C01811=1033.680,159.526,-103.122,169.533,42.942,158.097
C01812=1033.686,159.775,-103.145,169.536,42.941,158.097
C01813=1033.692,160.024,-103.167,169.539,42.940,158.097
C01814=1033.698,160.273,-103.190,169.542,42.939,158.097
C01815=1033.703,160.521,-103.212,169.544,42.939,158.097
C01816=1033.709,160.770,-103.235,169.547,42.938,158.097
C01817=1033.715,161.019,-103.257,169.550,42.937,158.097
C01818=1033.721,161.268,-103.280,169.553,42.936,158.097
C01819=1033.727,161.517,-103.303,169.556,42.935,158.097
C01820=1033.732,161.766,-103.326,169.559,42.934,158.097
C01821=1033.739,162.014,-103.348,169.561,42.933,158.097
C01822=1033.744,162.264,-103.370,169.564,42.933,158.097
C01823=1033.750,162.513,-103.393,169.566,42.932,158.097
C01824=1033.756,162.762,-103.416,169.569,42.931,158.097
C01825=1033.762,163.010,-103.438,169.572,42.930,158.097
C01826=1033.768,163.259,-103.461,169.575,42.930,158.097
C01827=1033.774,163.508,-103.484,169.577,42.929,158.097
C01828=1033.779,163.757,-103.507,169.580,42.928,158.098
C01829=1033.786,164.006,-103.530,169.583,42.927,158.098
C01830=1033.791,164.254,-103.552,169.586,42.926,158.098
C01831=1033.797,164.504,-103.575,169.589,42.925,158.098
C01832=1033.803,164.753,-103.598,169.592,42.924,158.098
C01833=1033.809,165.001,-103.620,169.595,42.924,158.098
C01834=1033.815,165.250,-103.643,169.598,42.922,158.098
C01835=1033.821,165.499,-103.666,169.600,42.922,158.098
C01836=1033.826,165.748,-103.689,169.603,42.921,158.098
C01837=1033.833,165.997,-103.711,169.606,42.920,158.098
C01838=1033.839,166.246,-103.735,169.608,42.919,158.098
C01839=1033.845,166.495,-103.757,169.611,42.918,158.098
C01840=1033.851,166.744,-103.780,169.614,42.918,158.098
C01841=1033.856,166.993,-103.803,169.617,42.916,158.098
C01842=1033.863,167.242,-103.826,169.620,42.916,158.098
C01843=1033.868,167.491,-103.849,169.623,42.915,158.098
C01844=1033.874,167.739,-103.872,169.626,42.914,158.098
C01845=1033.880,167.988,-103.895,169.628,42.913,158.098
C01846=1033.886,168.237,-103.917,169.631,42.913,158.098
C01847=1033.892,168.486,-103.940,169.634,42.912,158.098
C01848=1033.898,168.735,-103.963,169.637,42.911,158.098
C01849=1033.905,168.984,-103.987,169.640,42.910,158.098
C01850=1033.910,169.233,-104.010,169.643,42.910,158.098
C01851=1033.917,169.481,-104.032,169.645,42.908,158.098
C01852=1033.922,169.730,-104.055,169.649,42.908,158.099
C01853=1033.928,169.979,-104.078,169.651,42.907,158.099
C01854=1033.934,170.228,-104.101,169.654,42.906,158.099
C01855=1033.940,170.477,-104.124,169.657,42.905,158.099
C01856=1033.947,170.726,-104.147,169.660,42.904,158.099
C01857=1033.953,170.974,-104.170,169.663,42.903,158.099
C01858=1033.958,171.223,-104.193,169.666,42.902,158.099
C01859=1033.964,171.472,-104.216,169.669,42.902,158.099
C01860=1033.970,171.721,-104.239,169.672,42.901,158.099
C01861=1033.976,171.971,-104.262,169.675,42.900,158.099
C01862=1033.983,172.219,-104.285,169.678,42.899,158.099
C01863=1033.989,172.503,-104.312,169.681,42.898,158.099
C01864=1033.996,172.787,-104.338,169.684,42.897,158.099
C01865=1034.004,173.072,-104.364,169.688,42.897,158.099
C01866=1034.010,173.356,-104.391,169.690,42.896,158.099
C01867=1034.016,173.605,-104.414,169.693,42.894,158.099
C01868=1034.023,173.854,-104.436,169.696,42.894,158.099
C01869=1034.029,174.103,-104.461,169.699,42.893,158.099
C01870=1034.035,174.352,-104.483,169.702,42.892,158.099
C01871=1034.041,174.601,-104.506,169.705,42.891,158.099
C01872=1034.046,174.850,-104.529,169.708,42.891,158.100
C01873=1034.054,175.098,-104.553,169.711,42.889,158.100
C01874=1034.059,175.347,-104.576,169.714,42.889,158.100
C01875=1034.065,175.596,-104.599,169.717,42.888,158.100
C01876=1034.072,175.845,-104.623,169.720,42.887,158.100
C01877=1034.078,176.094,-104.646,169.723,42.886,158.100
C01878=1034.083,176.343,-104.669,169.726,42.886,158.100
C01879=1034.090,176.591,-104.692,169.729,42.884,158.100
C01880=1034.096,176.840,-104.715,169.732,42.884,158.100
C01881=1034.102,177.089,-104.739,169.735,42.883,158.100
C01882=1034.108,177.338,-104.762,169.738,42.882,158.100
C01883=1034.114,177.587,-104.785,169.741,42.882,158.100
C01884=1034.121,177.835,-104.809,169.744,42.881,158.100
C01885=1034.126,178.084,-104.831,169.747,42.880,158.100
C01886=1034.134,178.333,-104.855,169.750,42.879,158.100
C01887=1034.139,178.582,-104.878,169.753,42.878,158.100
C01888=1034.146,178.832,-104.901,169.756,42.877,158.100
C01889=1034.152,179.080,-104.925,169.759,42.877,158.101
C01890=1034.157,179.329,-104.948,169.762,42.876,158.101
C01891=1034.164,179.578,-104.972,169.765,42.875,158.101
C01892=1034.171,179.826,-104.994,169.768,42.874,158.101
C01893=1034.177,180.075,-105.018,169.771,42.873,158.101
C01894=1034.183,180.324,-105.041,169.774,42.872,158.101
C01895=1034.189,180.572,-105.065,169.777,42.872,158.101
C01896=1034.195,180.822,-105.088,169.780,42.871,158.101
C01897=1034.201,181.070,-105.112,169.783,42.870,158.101
C01898=1034.208,181.320,-105.135,169.787,42.869,158.101
C01899=1034.214,181.568,-105.159,169.790,42.868,158.101
C01900=1034.221,181.817,-105.182,169.793,42.868,158.101
C01901=1034.227,182.066,-105.205,169.795,42.867,158.101
C01902=1034.233,182.314,-105.229,169.798,42.866,158.101
C01903=1034.239,182.564,-105.252,169.801,42.865,158.101
C01904=1034.245,182.812,-105.276,169.804,42.865,158.101
C01905=1034.252,183.061,-105.300,169.807,42.864,158.102
C01906=1034.258,183.310,-105.323,169.810,42.863,158.101
C01907=1034.264,183.559,-105.347,169.813,42.862,158.102
C01908=1034.270,183.807,-105.371,169.817,42.862,158.102
C01909=1034.276,184.056,-105.395,169.820,42.861,158.102
C01910=1034.281,184.305,-105.419,169.823,42.861,158.102
C01911=1034.287,184.554,-105.442,169.826,42.860,158.102
C01912=1034.293,184.803,-105.467,169.829,42.859,158.102
C01913=1034.299,185.051,-105.491,169.832,42.859,158.102
C01914=1034.305,185.300,-105.514,169.835,42.858,158.102
C01915=1034.311,185.549,-105.539,169.838,42.858,158.102
C01916=1034.317,185.797,-105.562,169.841,42.857,158.103
C01917=1034.323,186.046,-105.587,169.844,42.857,158.103
C01918=1034.329,186.295,-105.611,169.848,42.856,158.103
C01919=1034.335,186.544,-105.635,169.851,42.856,158.103
C01920=1034.341,186.792,-105.659,169.854,42.855,158.103
C01921=1034.346,187.041,-105.683,169.857,42.855,158.103
C01922=1034.353,187.290,-105.707,169.859,42.853,158.103
C01923=1034.358,187.539,-105.731,169.863,42.853,158.103
C01924=1034.365,187.788,-105.755,169.867,42.852,158.103
C01925=1034.371,188.036,-105.779,169.870,42.852,158.104
C01926=1034.376,188.286,-105.803,169.873,42.851,158.104
C01927=1034.383,188.569,-105.831,169.876,42.851,158.104
C01928=1034.390,188.853,-105.859,169.880,42.850,158.104
C01929=1034.397,189.137,-105.886,169.883,42.850,158.104
C01930=1034.404,189.421,-105.914,169.887,42.849,158.104
C01931=1034.410,189.670,-105.938,169.890,42.848,158.104
C01932=1034.416,189.919,-105.962,169.893,42.848,158.105
C01933=1034.422,190.168,-105.986,169.896,42.847,158.105
C01934=1034.428,190.416,-106.010,169.899,42.846,158.105
C01935=1034.434,190.665,-106.034,169.903,42.846,158.105
C01936=1034.440,190.914,-106.059,169.906,42.845,158.105
C01937=1034.447,191.162,-106.083,169.909,42.845,158.105
C01938=1034.452,191.411,-106.108,169.912,42.844,158.105
C01939=1034.459,191.660,-106.132,169.915,42.844,158.105
C01940=1034.464,191.909,-106.156,169.918,42.843,158.105
C01941=1034.470,192.157,-106.180,169.921,42.843,158.106
C01942=1034.476,192.406,-106.204,169.925,42.842,158.106
C01943=1034.483,192.654,-106.229,169.928,42.841,158.106
C01944=1034.489,192.903,-106.253,169.931,42.841,158.106
C01945=1034.495,193.152,-106.277,169.934,42.840,158.106
C01946=1034.501,193.401,-106.302,169.937,42.840,158.106
C01947=1034.507,193.650,-106.326,169.940,42.839,158.106
C01948=1034.513,193.899,-106.351,169.944,42.839,158.106
C01949=1034.519,194.147,-106.375,169.947,42.838,158.107
C01950=1034.525,194.396,-106.399,169.950,42.838,158.107
C01951=1034.532,194.645,-106.423,169.954,42.837,158.107
C01952=1034.538,194.893,-106.448,169.957,42.837,158.107
C01953=1034.544,195.142,-106.472,169.961,42.836,158.107
C01954=1034.550,195.391,-106.497,169.964,42.836,158.107
C01955=1034.556,195.639,-106.521,169.967,42.835,158.107
C01956=1034.562,195.888,-106.546,169.970,42.835,158.107
C01957=1034.569,196.137,-106.570,169.973,42.834,158.108
C01958=1034.575,196.385,-106.595,169.977,42.833,158.108
C01959=1034.581,196.634,-106.619,169.980,42.833,158.108
C01960=1034.587,196.884,-106.644,169.983,42.832,158.108
C01961=1034.593,197.131,-106.668,169.986,42.832,158.108
C01962=1034.599,197.381,-106.693,169.990,42.831,158.108
C01963=1034.606,197.630,-106.717,169.993,42.831,158.108
C01964=1034.612,197.878,-106.742,169.996,42.830,158.109
C01965=1034.618,198.126,-106.766,169.999,42.830,158.109
C01966=1034.624,198.375,-106.791,170.003,42.829,158.109
C01967=1034.630,198.624,-106.816,170.006,42.829,158.109
C01968=1034.637,198.873,-106.840,170.009,42.828,158.109
C01969=1034.643,199.122,-106.865,170.012,42.828,158.109
C01970=1034.649,199.370,-106.889,170.016,42.827,158.109
C01971=1034.655,199.619,-106.914,170.019,42.826,158.109
C01972=1034.662,199.868,-106.938,170.023,42.827,158.110
C01973=1034.668,200.117,-106.963,170.026,42.826,158.110
C01974=1034.675,200.366,-106.987,170.030,42.825,158.110
C01975=1034.681,200.614,-107.012,170.033,42.825,158.110
C01976=1034.687,200.862,-107.038,170.036,42.824,158.110
C01977=1034.693,201.112,-107.062,170.039,42.824,158.110
C01978=1034.700,201.360,-107.087,170.043,42.824,158.111
C01979=1034.705,201.609,-107.112,170.046,42.823,158.111
C01980=1034.711,201.857,-107.137,170.049,42.823,158.111
C01981=1034.717,202.106,-107.162,170.052,42.822,158.111
C01982=1034.723,202.354,-107.187,170.056,42.822,158.111
C01983=1034.729,202.604,-107.212,170.059,42.822,158.111
C01984=1034.736,202.852,-107.237,170.062,42.821,158.112
C01985=1034.741,203.100,-107.262,170.067,42.821,158.112
C01986=1034.747,203.350,-107.287,170.070,42.821,158.112
C01987=1034.754,203.598,-107.312,170.073,42.820,158.112
C01988=1034.760,203.847,-107.337,170.076,42.820,158.112
C01989=1034.766,204.095,-107.362,170.080,42.820,158.113
C01990=1034.773,204.344,-107.388,170.083,42.819,158.113
C01991=1034.798,205.393,-107.493,170.407,42.924,158.158
C01992=1034.808,205.731,-107.529,170.411,42.924,158.159
C01993=1034.817,206.069,-107.565,170.414,42.925,158.159
C01994=1034.826,206.405,-107.600,170.417,42.925,158.159
C01995=1034.835,206.743,-107.636,170.421,42.925,158.160
C01996=1034.842,206.992,-107.663,170.423,42.926,158.160
C01997=1034.848,207.240,-107.689,170.425,42.927,158.160
C01998=1034.855,207.489,-107.716,170.427,42.927,158.160
C01999=1034.862,207.737,-107.742,170.430,42.927,158.161
C02000=1034.869,207.985,-107.768,170.432,42.928,158.161
C02001=1034.875,208.235,-107.795,170.435,42.928,158.161
C02002=1034.882,208.483,-107.821,170.438,42.929,158.162
C02003=1034.889,208.731,-107.848,170.440,42.929,158.162
C02004=1034.896,208.979,-107.875,170.442,42.929,158.162
C02005=1034.902,209.228,-107.902,170.445,42.930,158.162
C02006=1034.909,209.477,-107.928,170.448,42.930,158.163
C02007=1034.916,209.725,-107.954,170.450,42.931,158.163
C02008=1034.922,209.974,-107.981,170.452,42.931,158.163
C02009=1034.929,210.222,-108.007,170.455,42.932,158.163
C02010=1034.936,210.470,-108.034,170.457,42.932,158.164
C02011=1034.942,210.719,-108.061,170.460,42.932,158.164
C02012=1034.950,210.968,-108.088,170.463,42.933,158.164
C02013=1034.956,211.216,-108.114,170.465,42.933,158.165
C02014=1034.962,211.465,-108.141,170.467,42.934,158.165
C02015=1034.970,211.713,-108.168,170.469,42.934,158.165
C02016=1034.976,211.961,-108.195,170.473,42.935,158.165
C02017=1034.983,212.210,-108.221,170.475,42.935,158.166
C02018=1034.989,212.458,-108.249,170.477,42.935,158.166
C02019=1034.996,212.707,-108.275,170.480,42.936,158.166
C02020=1035.002,212.956,-108.302,170.482,42.936,158.166
C02021=1035.010,213.204,-108.329,170.485,42.937,158.167
C02022=1035.015,213.452,-108.356,170.488,42.938,158.167
C02023=1035.022,213.701,-108.383,170.490,42.938,158.167
C02024=1035.029,213.949,-108.410,170.492,42.938,158.168
C02025=1035.036,214.198,-108.437,170.494,42.939,158.168
C02026=1035.042,214.446,-108.463,170.498,42.939,158.168
C02027=1035.049,214.695,-108.490,170.500,42.939,158.168
C02028=1035.056,214.944,-108.517,170.502,42.940,158.169
C02029=1035.062,215.191,-108.544,170.505,42.941,158.169
C02030=1035.069,215.440,-108.571,170.508,42.941,158.169
C02031=1035.076,215.688,-108.598,170.510,42.942,158.170
C02032=1035.083,215.937,-108.625,170.513,42.942,158.170
C02033=1035.089,216.185,-108.652,170.515,42.942,158.170
C02034=1035.096,216.434,-108.679,170.518,42.943,158.171
C02035=1035.103,216.683,-108.706,170.520,42.943,158.171
C02036=1035.110,216.931,-108.733,170.523,42.944,158.171
C02037=1035.116,217.180,-108.760,170.525,42.944,158.171
C02038=1035.123,217.427,-108.787,170.528,42.945,158.172
C02039=1035.130,217.676,-108.814,170.531,42.945,158.172
C02040=1035.137,217.925,-108.841,170.533,42.945,158.172
C02041=1035.143,218.174,-108.868,170.536,42.946,158.173
C02042=1035.150,218.422,-108.895,170.539,42.946,158.173
C02043=1035.157,218.670,-108.922,170.541,42.947,158.173
C02044=1035.163,218.919,-108.949,170.543,42.947,158.173
C02045=1035.171,219.167,-108.976,170.546,42.948,158.174
C02046=1035.177,219.416,-109.003,170.549,42.948,158.174
C02047=1035.184,219.664,-109.031,170.551,42.949,158.174
C02048=1035.193,220.007,-109.068,170.556,42.949,158.175
C02049=1035.202,220.349,-109.106,170.559,42.950,158.175
C02050=1035.212,220.693,-109.144,170.562,42.951,158.176
C02051=1035.220,221.036,-109.181,170.566,42.952,158.176
C02052=1035.227,221.284,-109.209,170.568,42.952,158.176
C02053=1035.234,221.532,-109.236,170.571,42.952,158.176
C02054=1035.241,221.781,-109.263,170.574,42.953,158.177
C02055=1035.247,222.029,-109.290,170.576,42.953,158.177
C02056=1035.254,222.277,-109.318,170.579,42.954,158.177
C02057=1035.260,222.526,-109.346,170.582,42.954,158.178
C02058=1035.267,222.775,-109.373,170.584,42.955,158.178
C02059=1035.273,223.023,-109.400,170.586,42.955,158.178
C02060=1035.281,223.271,-109.428,170.590,42.956,158.179
C02061=1035.287,223.520,-109.455,170.592,42.956,158.179
C02062=1035.293,223.768,-109.482,170.594,42.957,158.179
C02063=1035.300,224.017,-109.510,170.598,42.957,158.180
C02064=1035.307,224.265,-109.537,170.600,42.958,158.180
C02065=1035.314,224.513,-109.565,170.602,42.959,158.180
C02066=1035.321,224.762,-109.592,170.606,42.959,158.180
C02067=1035.327,225.010,-109.620,170.608,42.959,158.181
C02068=1035.334,225.259,-109.647,170.610,42.960,158.181
C02069=1035.340,225.508,-109.675,170.614,42.960,158.181
C02070=1035.347,225.756,-109.702,170.616,42.961,158.182
C02071=1035.355,226.004,-109.730,170.618,42.961,158.182
C02072=1035.361,226.253,-109.757,170.622,42.962,158.182
C02073=1035.367,226.500,-109.785,170.624,42.962,158.183
C02074=1035.374,226.749,-109.812,170.627,42.962,158.183
C02075=1035.381,226.997,-109.840,170.630,42.963,158.183
C02076=1035.387,227.246,-109.868,170.632,42.964,158.183
C02077=1035.395,227.494,-109.895,170.635,42.964,158.184
C02078=1035.401,227.742,-109.923,170.638,42.965,158.184
C02079=1035.408,227.991,-109.950,170.640,42.966,158.184
C02080=1035.415,228.239,-109.978,170.643,42.966,158.185
C02081=1035.421,228.488,-110.006,170.646,42.967,158.185
C02082=1035.428,228.736,-110.034,170.649,42.967,158.185
C02083=1035.435,228.985,-110.061,170.651,42.968,158.186
C02084=1035.442,229.233,-110.089,170.654,42.968,158.186
C02085=1035.448,229.481,-110.117,170.657,42.969,158.186
C02086=1035.455,229.730,-110.145,170.659,42.969,158.187
C02087=1035.461,229.979,-110.173,170.662,42.970,158.187
C02088=1035.467,230.227,-110.201,170.665,42.970,158.187
C02089=1035.474,230.475,-110.228,170.667,42.971,158.188
C02090=1035.481,230.723,-110.257,170.671,42.972,158.188
C02091=1035.488,230.972,-110.285,170.673,42.972,158.188
C02092=1035.495,231.220,-110.312,170.676,42.973,158.189
C02093=1035.501,231.469,-110.340,170.679,42.973,158.189
C02094=1035.508,231.717,-110.368,170.681,42.974,158.189
C02095=1035.515,231.966,-110.395,170.685,42.974,158.190
C02096=1035.521,232.214,-110.425,170.687,42.975,158.190
C02097=1035.527,232.462,-110.452,170.689,42.976,158.190
C02098=1035.534,232.711,-110.480,170.693,42.976,158.191
C02099=1035.541,232.959,-110.508,170.695,42.977,158.191
C02100=1035.548,233.207,-110.536,170.698,42.977,158.191
C02101=1035.554,233.456,-110.564,170.701,42.978,158.192
C02102=1035.560,233.704,-110.592,170.703,42.979,158.192
C02103=1035.567,233.952,-110.621,170.706,42.979,158.192
C02104=1035.576,234.288,-110.658,170.710,42.980,158.193
C02105=1035.585,234.623,-110.697,170.714,42.981,158.193
C02106=1035.594,234.958,-110.735,170.718,42.981,158.194
C02107=1035.604,235.293,-110.772,170.721,42.982,158.194
C02108=1035.610,235.542,-110.801,170.724,42.983,158.194
C02109=1035.616,235.790,-110.828,170.727,42.983,158.195
C02110=1035.623,236.038,-110.857,170.730,42.984,158.195
C02111=1035.631,236.287,-110.885,170.733,42.984,158.195
C02112=1035.636,236.536,-110.913,170.735,42.985,158.196
C02113=1035.643,236.784,-110.942,170.739,42.986,158.196
C02114=1035.650,237.032,-110.969,170.741,42.986,158.196
C02115=1035.657,237.280,-110.998,170.744,42.987,158.197
C02116=1035.663,237.529,-111.026,170.747,42.987,158.197
C02117=1035.670,237.777,-111.055,170.750,42.988,158.198
C02118=1035.677,238.025,-111.082,170.753,42.989,158.198
C02119=1035.684,238.274,-111.111,170.756,42.989,158.198
C02120=1035.690,238.522,-111.140,170.758,42.990,158.199
C02121=1035.697,238.770,-111.168,170.762,42.991,158.199
C02122=1035.704,239.019,-111.196,170.764,42.991,158.199
C02123=1035.710,239.267,-111.225,170.767,42.992,158.200
C02124=1035.717,239.515,-111.252,170.770,42.993,158.200
C02125=1035.724,239.763,-111.281,170.773,42.993,158.200
C02126=1035.730,240.013,-111.310,170.776,42.994,158.201
C02127=1035.737,240.260,-111.338,170.779,42.994,158.201
C02128=1035.744,240.508,-111.367,170.781,42.995,158.201
C02129=1035.750,240.757,-111.395,170.785,42.995,158.202
C02130=1035.757,241.005,-111.423,170.787,42.996,158.202
C02131=1035.764,241.253,-111.452,170.790,42.996,158.202
C02132=1035.771,241.502,-111.480,170.793,42.997,158.203
C02133=1035.777,241.750,-111.509,170.796,42.998,158.203
C02134=1035.784,241.998,-111.538,170.799,42.999,158.204
C02135=1035.790,242.247,-111.566,170.802,42.999,158.204
C02136=1035.797,242.495,-111.595,170.804,43.000,158.204
C02137=1035.804,242.743,-111.624,170.808,43.001,158.205
C02138=1035.810,242.992,-111.653,170.810,43.001,158.205
C02139=1035.817,243.239,-111.682,170.814,43.002,158.205
C02140=1035.823,243.488,-111.710,170.816,43.002,158.206
C02141=1035.830,243.736,-111.738,170.819,43.003,158.206
C02142=1035.837,243.985,-111.768,170.822,43.004,158.206
C02143=1035.844,244.233,-111.796,170.825,43.005,158.207
C02144=1035.850,244.481,-111.825,170.828,43.005,158.207
C02145=1035.857,244.729,-111.853,170.831,43.006,158.207
C02146=1035.863,244.977,-111.882,170.833,43.007,158.208
C02147=1035.870,245.226,-111.911,170.837,43.008,158.208
C02148=1035.876,245.474,-111.940,170.839,43.008,158.209
C02149=1035.882,245.722,-111.969,170.843,43.009,158.209
C02150=1035.889,245.970,-111.998,170.845,43.010,158.209
C02151=1035.896,246.219,-112.027,170.849,43.011,158.210
C02152=1035.902,246.467,-112.056,170.851,43.011,158.210
C02153=1035.909,246.715,-112.085,170.854,43.012,158.211
C02154=1035.915,246.963,-112.114,170.857,43.013,158.211
C02155=1035.921,247.212,-112.143,170.860,43.013,158.211
C02156=1035.929,247.460,-112.172,170.864,43.014,158.212
C02157=1035.935,247.708,-112.201,170.866,43.015,158.212
C02158=1035.941,247.956,-112.230,170.870,43.016,158.213
C02159=1035.948,248.205,-112.260,170.872,43.017,158.213
C02160=1035.957,248.535,-112.299,170.877,43.017,158.213
C02161=1035.965,248.864,-112.337,170.880,43.019,158.214
C02162=1035.974,249.193,-112.376,170.884,43.019,158.214
C02163=1035.983,249.522,-112.414,170.888,43.020,158.215
C02164=1035.990,249.771,-112.444,170.891,43.021,158.215
C02165=1035.996,250.019,-112.473,170.894,43.022,158.216
C02166=1036.002,250.267,-112.502,170.898,43.023,158.216
C02167=1036.009,250.516,-112.531,170.900,43.024,158.217
C02168=1036.016,250.764,-112.560,170.904,43.024,158.217
C02169=1036.023,251.012,-112.589,170.906,43.025,158.217
C02170=1036.030,251.260,-112.619,170.909,43.025,158.218
C02171=1036.036,251.508,-112.648,170.913,43.026,158.218
C02172=1036.043,251.757,-112.677,170.915,43.027,158.218
C02173=1036.049,252.005,-112.706,170.919,43.028,158.219
C02174=1036.056,252.253,-112.736,170.921,43.029,158.219
C02175=1036.063,252.501,-112.765,170.925,43.029,158.220
C02176=1036.069,252.749,-112.794,170.928,43.030,158.220
C02177=1036.076,252.998,-112.823,170.930,43.031,158.220
C02178=1036.083,253.246,-112.853,170.934,43.032,158.221
C02179=1036.089,253.494,-112.882,170.937,43.032,158.221
C02180=1036.096,253.743,-112.912,170.940,43.033,158.222
C02181=1036.103,253.990,-112.941,170.943,43.034,158.222
C02182=1036.109,254.239,-112.971,170.947,43.035,158.223
C02183=1036.116,254.487,-112.999,170.949,43.036,158.223
C02184=1036.123,254.734,-113.029,170.953,43.036,158.223
C02185=1036.130,254.983,-113.058,170.956,43.037,158.224
C02186=1036.136,255.231,-113.087,170.959,43.038,158.224
C02187=1036.143,255.480,-113.118,170.962,43.039,158.225
C02188=1036.149,255.728,-113.147,170.965,43.040,158.225
C02189=1036.157,255.976,-113.177,170.968,43.040,158.225
C02190=1036.164,256.224,-113.205,170.971,43.041,158.226
C02191=1036.170,256.473,-113.235,170.975,43.041,158.226
C02192=1036.177,256.720,-113.264,170.977,43.042,158.226
C02193=1036.184,256.969,-113.294,170.981,43.043,158.227
C02194=1036.190,257.217,-113.324,170.984,43.044,158.227
C02195=1036.197,257.465,-113.353,170.986,43.044,158.228
C02196=1036.204,257.713,-113.383,170.990,43.045,158.228
C02197=1036.211,257.962,-113.412,170.993,43.046,158.228
C02198=1036.217,258.209,-113.442,170.996,43.047,158.229
C02199=1036.225,258.458,-113.471,170.999,43.048,158.229
C02200=1036.232,258.706,-113.501,171.003,43.048,158.230
C02201=1036.238,258.954,-113.530,171.006,43.049,158.230
C02202=1036.245,259.202,-113.560,171.009,43.050,158.230
C02203=1036.252,259.450,-113.589,171.012,43.051,158.231
C02204=1036.259,259.699,-113.619,171.015,43.051,158.231
C02205=1036.266,259.947,-113.649,171.019,43.052,158.232
C02206=1036.272,260.195,-113.678,171.021,43.053,158.232
C02207=1036.279,260.443,-113.708,171.025,43.054,158.233
C02208=1036.286,260.691,-113.737,171.028,43.054,158.233
C02209=1036.293,260.939,-113.767,171.032,43.055,158.233
C02210=1036.301,261.187,-113.797,171.034,43.056,158.234
C02211=1036.307,261.436,-113.826,171.038,43.057,158.234
C02212=1036.314,261.684,-113.856,171.041,43.057,158.235
C02213=1036.321,261.931,-113.886,171.045,43.059,158.235
C02214=1036.327,262.180,-113.917,171.047,43.060,158.236
C02215=1036.334,262.429,-113.946,171.051,43.060,158.236
C02216=1036.342,262.756,-113.986,171.055,43.061,158.237
C02217=1036.351,263.084,-114.025,171.059,43.063,158.237
C02218=1036.360,263.413,-114.065,171.064,43.064,158.238
C02219=1036.369,263.741,-114.105,171.068,43.065,158.238
C02220=1036.376,263.989,-114.135,171.071,43.066,158.239
C02221=1036.382,264.236,-114.165,171.074,43.067,158.239
C02222=1036.389,264.485,-114.196,171.078,43.067,158.240
C02223=1036.396,264.733,-114.226,171.081,43.069,158.240
C02224=1036.403,264.981,-114.255,171.084,43.070,158.241
C02225=1036.409,265.229,-114.286,171.087,43.070,158.241
C02226=1036.416,265.477,-114.316,171.091,43.071,158.241
C02227=1036.423,265.725,-114.346,171.094,43.072,158.242
C02228=1036.429,265.974,-114.377,171.098,43.073,158.242
C02229=1036.436,266.222,-114.407,171.100,43.074,158.243
C02230=1036.443,266.469,-114.437,171.104,43.075,158.243
C02231=1036.450,266.717,-114.467,171.107,43.075,158.244
C02232=1036.456,266.966,-114.497,171.111,43.077,158.244
C02233=1036.463,267.213,-114.527,171.113,43.078,158.245
C02234=1036.469,267.462,-114.558,171.117,43.078,158.245
C02235=1036.476,267.710,-114.588,171.121,43.080,158.246
C02236=1036.484,267.958,-114.618,171.124,43.080,158.246
C02237=1036.489,268.206,-114.649,171.127,43.081,158.246
C02238=1036.497,268.454,-114.679,171.130,43.083,158.247
C02239=1036.503,268.702,-114.710,171.134,43.083,158.247
C02240=1036.510,268.950,-114.740,171.137,43.084,158.248
C02241=1036.516,269.198,-114.771,171.141,43.085,158.248
C02242=1036.523,269.447,-114.801,171.144,43.086,158.249
C02243=1036.530,269.695,-114.831,171.148,43.087,158.249
C02244=1036.537,269.942,-114.862,171.150,43.088,158.250
C02245=1036.543,270.191,-114.893,171.154,43.089,158.250
C02246=1036.550,270.439,-114.923,171.157,43.090,158.251
C02247=1036.557,270.687,-114.953,171.161,43.091,158.251
C02248=1036.564,270.934,-114.984,171.164,43.092,158.252
C02249=1036.571,271.182,-115.014,171.168,43.093,158.252
C02250=1036.577,271.431,-115.045,171.170,43.094,158.252
C02251=1036.584,271.679,-115.076,171.174,43.095,158.253
C02252=1036.590,271.926,-115.106,171.178,43.096,158.253
C02253=1036.597,272.175,-115.137,171.181,43.097,158.254
C02254=1036.604,272.423,-115.168,171.185,43.098,158.254
C02255=1036.611,272.671,-115.198,171.188,43.099,158.255
C02256=1036.617,272.919,-115.230,171.192,43.100,158.255
C02257=1036.624,273.166,-115.259,171.194,43.101,158.256
C02258=1036.631,273.414,-115.291,171.198,43.102,158.256
C02259=1036.637,273.663,-115.322,171.201,43.103,158.257
C02260=1036.644,273.911,-115.352,171.205,43.104,158.257
C02261=1036.651,274.159,-115.383,171.209,43.105,158.258
C02262=1036.657,274.407,-115.414,171.212,43.106,158.258
C02263=1036.664,274.654,-115.444,171.216,43.107,158.259
C02264=1036.671,274.902,-115.476,171.219,43.108,158.259
C02265=1036.677,275.151,-115.506,171.222,43.109,158.260
C02266=1036.685,275.398,-115.537,171.225,43.110,158.260
C02267=1036.691,275.647,-115.568,171.229,43.111,158.261
C02268=1036.698,275.895,-115.599,171.233,43.113,158.261
C02269=1036.705,276.143,-115.630,171.236,43.113,158.262
C02270=1036.712,276.391,-115.661,171.240,43.115,158.262
C02271=1036.718,276.638,-115.692,171.243,43.115,158.263
C02272=1036.727,276.972,-115.733,171.248,43.117,158.264
C02273=1036.737,277.305,-115.775,171.253,43.118,158.264
C02274=1036.746,277.637,-115.817,171.257,43.119,158.265
C02275=1036.755,277.970,-115.858,171.262,43.121,158.266
C02276=1036.762,278.218,-115.889,171.265,43.122,158.266
C02277=1036.768,278.466,-115.921,171.269,43.123,158.267
C02278=1036.775,278.714,-115.952,171.272,43.125,158.267
C02279=1036.781,278.961,-115.983,171.276,43.125,158.268
C02280=1036.788,279.209,-116.015,171.279,43.127,158.268
C02281=1036.794,279.458,-116.045,171.283,43.128,158.269
C02282=1036.801,279.705,-116.077,171.286,43.129,158.269
C02283=1036.808,279.953,-116.108,171.290,43.130,158.270
C02284=1036.815,280.201,-116.140,171.294,43.131,158.270
C02285=1036.821,280.449,-116.171,171.297,43.133,158.271
C02286=1036.829,280.697,-116.202,171.301,43.133,158.271
C02287=1036.835,280.945,-116.233,171.305,43.135,158.272
C02288=1036.842,281.193,-116.265,171.308,43.136,158.272
C02289=1036.849,281.440,-116.296,171.312,43.137,158.273
C02290=1036.856,281.688,-116.328,171.315,43.138,158.273
C02291=1036.862,281.936,-116.359,171.319,43.139,158.274
C02292=1036.869,282.184,-116.390,171.323,43.141,158.275
C02293=1036.876,282.432,-116.422,171.326,43.141,158.275
C02294=1036.883,282.680,-116.453,171.330,43.143,158.276
C02295=1036.889,282.928,-116.485,171.334,43.144,158.276
C02296=1036.896,283.176,-116.516,171.336,43.146,158.277
C02297=1036.903,283.424,-116.548,171.340,43.146,158.277
C02298=1036.909,283.672,-116.579,171.343,43.148,158.278
C02299=1036.916,283.920,-116.610,171.348,43.149,158.278
C02300=1036.923,284.167,-116.642,171.352,43.150,158.279
C02301=1036.930,284.416,-116.674,171.355,43.151,158.279
C02302=1036.937,284.664,-116.705,171.359,43.152,158.280
C02303=1036.944,284.912,-116.737,171.363,43.153,158.280
C02304=1036.951,285.159,-116.769,171.366,43.155,158.281
C02305=1036.957,285.407,-116.800,171.370,43.156,158.282
C02306=1036.964,285.655,-116.832,171.373,43.157,158.282
C02307=1036.971,285.903,-116.863,171.377,43.158,158.283
C02308=1036.978,286.151,-116.894,171.381,43.159,158.283
C02309=1036.985,286.399,-116.926,171.384,43.161,158.284
C02310=1036.992,286.647,-116.958,171.388,43.162,158.284
C02311=1036.999,286.895,-116.990,171.392,43.163,158.285
C02312=1037.005,287.142,-117.021,171.395,43.164,158.285
C02313=1037.012,287.390,-117.054,171.399,43.165,158.286
C02314=1037.018,287.638,-117.085,171.403,43.166,158.286
C02315=1037.025,287.886,-117.117,171.406,43.168,158.287
C02316=1037.032,288.133,-117.149,171.410,43.169,158.288
C02317=1037.039,288.382,-117.181,171.414,43.170,158.288
C02318=1037.046,288.629,-117.214,171.417,43.172,158.289
C02319=1037.052,288.877,-117.245,171.421,43.173,158.289
C02320=1037.059,289.125,-117.276,171.425,43.174,158.290
C02321=1037.066,289.372,-117.309,171.428,43.176,158.290
C02322=1037.074,289.621,-117.340,171.433,43.177,158.291
C02323=1037.080,289.869,-117.373,171.437,43.178,158.292
C02324=1037.087,290.116,-117.405,171.440,43.179,158.292
C02325=1037.094,290.364,-117.437,171.444,43.181,158.293
C02326=1037.100,290.612,-117.469,171.448,43.182,158.293
C02327=1037.107,290.860,-117.501,171.451,43.183,158.294
C02328=1037.117,291.205,-117.545,171.456,43.185,158.295
C02329=1037.126,291.549,-117.590,171.462,43.187,158.296
C02330=1037.136,291.894,-117.635,171.467,43.189,158.296
C02331=1037.145,292.238,-117.679,171.472,43.191,158.297
C02332=1037.152,292.487,-117.712,171.476,43.192,158.298
C02333=1037.159,292.734,-117.744,171.481,43.193,158.298
C02334=1037.166,292.982,-117.776,171.484,43.194,158.299
C02335=1037.173,293.230,-117.809,171.488,43.196,158.300
C02336=1037.180,293.477,-117.841,171.492,43.197,158.300
C02337=1037.186,293.726,-117.873,171.496,43.199,158.301
C02338=1037.193,293.974,-117.906,171.499,43.200,158.301
C02339=1037.200,294.221,-117.938,171.503,43.202,158.302
C02340=1037.207,294.468,-117.970,171.507,43.203,158.303
C02341=1037.213,294.716,-118.002,171.511,43.204,158.303
C02342=1037.220,294.965,-118.035,171.515,43.205,158.304
C02343=1037.227,295.212,-118.067,171.519,43.207,158.305
C02344=1037.234,295.460,-118.100,171.523,43.208,158.305
C02345=1037.241,295.708,-118.133,171.526,43.210,158.306
C02346=1037.248,295.955,-118.165,171.530,43.212,158.306
C02347=1037.254,296.203,-118.198,171.534,43.213,158.307
C02348=1037.261,296.451,-118.231,171.539,43.214,158.308
C02349=1037.267,296.699,-118.264,171.542,43.216,158.308
C02350=1037.274,296.946,-118.296,171.546,43.217,158.309
C02351=1037.281,297.194,-118.329,171.550,43.219,158.310
C02352=1037.287,297.442,-118.362,171.554,43.220,158.310
C02353=1037.294,297.689,-118.395,171.557,43.222,158.311
C02354=1037.301,297.937,-118.427,171.561,43.223,158.311
C02355=1037.307,298.185,-118.460,171.566,43.225,158.312
C02356=1037.314,298.432,-118.493,171.570,43.226,158.313
C02357=1037.321,298.680,-118.526,171.574,43.228,158.314
C02358=1037.328,298.927,-118.558,171.577,43.229,158.314
C02359=1037.335,299.176,-118.592,171.581,43.231,158.315
C02360=1037.341,299.423,-118.624,171.586,43.232,158.315
C02361=1037.347,299.671,-118.657,171.589,43.234,158.316
C02362=1037.355,299.918,-118.690,171.593,43.236,158.317
C02363=1037.362,300.166,-118.723,171.597,43.237,158.317
C02364=1037.369,300.414,-118.756,171.601,43.238,158.318
C02365=1037.375,300.662,-118.789,171.606,43.240,158.319
C02366=1037.382,300.909,-118.823,171.609,43.241,158.319
C02367=1037.389,301.157,-118.855,171.613,43.243,158.320
C02368=1037.396,301.405,-118.888,171.617,43.244,158.321
C02369=1037.402,301.653,-118.921,171.622,43.246,158.321
C02370=1037.409,301.900,-118.955,171.626,43.247,158.322
C02371=1037.417,302.148,-118.987,171.629,43.249,158.323
C02372=1037.423,302.396,-119.020,171.633,43.251,158.323
C02373=1037.430,302.643,-119.053,171.638,43.252,158.324
C02374=1037.437,302.891,-119.086,171.642,43.254,158.325
C02375=1037.444,303.138,-119.120,171.646,43.255,158.325
C02376=1037.451,303.386,-119.152,171.649,43.257,158.326
C02377=1037.457,303.634,-119.185,171.654,43.258,158.327
C02378=1037.465,303.881,-119.219,171.658,43.260,158.327
C02379=1037.471,304.129,-119.252,171.662,43.262,158.328
C02380=1037.478,304.377,-119.285,171.667,43.263,158.329
C02381=1037.486,304.625,-119.318,171.670,43.265,158.329
C02382=1037.492,304.872,-119.351,171.674,43.267,158.330
C02383=1037.499,305.120,-119.385,171.678,43.268,158.331
C02384=1037.510,305.481,-119.433,171.684,43.270,158.332
C02385=1037.519,305.843,-119.481,171.691,43.273,158.333
C02386=1037.530,306.204,-119.530,171.697,43.275,158.334
C02387=1037.540,306.566,-119.579,171.703,43.277,158.335
C02388=1037.547,306.813,-119.612,171.707,43.279,158.335
C02389=1037.555,307.060,-119.645,171.711,43.280,158.336
C02390=1037.561,307.309,-119.679,171.715,43.282,158.337
C02391=1037.568,307.556,-119.712,171.719,43.284,158.338
C02392=1037.575,307.803,-119.746,171.724,43.285,158.338
C02393=1037.582,308.051,-119.780,171.728,43.287,158.339
C02394=1037.589,308.299,-119.813,171.732,43.289,158.340
C02395=1037.597,308.546,-119.846,171.736,43.290,158.340
C02396=1037.604,308.794,-119.879,171.740,43.292,158.341
C02397=1037.611,309.042,-119.913,171.744,43.293,158.342
C02398=1037.618,309.290,-119.946,171.749,43.295,158.342
C02399=1037.625,309.537,-119.980,171.753,43.296,158.343
C02400=1037.632,309.784,-120.014,171.758,43.298,158.344
C02401=1037.640,310.032,-120.047,171.762,43.300,158.345
C02402=1037.647,310.280,-120.080,171.765,43.301,158.345
C02403=1037.654,310.528,-120.114,171.770,43.303,158.346
C02404=1037.660,310.775,-120.147,171.774,43.305,158.347
C02405=1037.668,311.022,-120.181,171.779,43.307,158.348
C02406=1037.675,311.270,-120.215,171.783,43.308,158.348
C02407=1037.683,311.517,-120.248,171.788,43.310,158.349
C02408=1037.690,311.765,-120.282,171.792,43.311,158.350
C02409=1037.697,312.013,-120.316,171.796,43.313,158.350
C02410=1037.703,312.260,-120.350,171.800,43.315,158.351
C02411=1037.710,312.508,-120.384,171.804,43.317,158.352
C02412=1037.717,312.756,-120.418,171.809,43.319,158.353
C02413=1037.724,313.003,-120.452,171.813,43.321,158.353
C02414=1037.731,313.250,-120.486,171.817,43.322,158.354
C02415=1037.737,313.498,-120.521,171.822,43.324,158.355
C02416=1037.744,313.745,-120.554,171.826,43.326,158.356
C02417=1037.751,313.993,-120.589,171.831,43.328,158.356
C02418=1037.758,314.240,-120.623,171.835,43.330,158.357
C02419=1037.765,314.488,-120.658,171.839,43.331,158.358
C02420=1037.772,314.736,-120.692,171.844,43.334,158.359
C02421=1037.778,314.983,-120.726,171.848,43.336,158.360
C02422=1037.785,315.230,-120.760,171.853,43.337,158.360
C02423=1037.793,315.478,-120.794,171.857,43.339,158.361
C02424=1037.799,315.725,-120.829,171.861,43.341,158.362
C02425=1037.807,315.973,-120.863,171.865,43.343,158.363
C02426=1037.813,316.221,-120.897,171.870,43.344,158.363
C02427=1037.821,316.468,-120.932,171.874,43.347,158.364
C02428=1037.827,316.716,-120.966,171.878,43.349,158.365
C02429=1037.835,316.963,-121.001,171.883,43.350,158.366
C02430=1037.841,317.211,-121.035,171.887,43.352,158.367
C02431=1037.848,317.459,-121.069,171.892,43.354,158.367
C02432=1037.856,317.706,-121.104,171.896,43.357,158.368
C02433=1037.862,317.954,-121.138,171.901,43.358,158.369
C02434=1037.870,318.201,-121.173,171.905,43.360,158.370
C02435=1037.876,318.449,-121.207,171.910,43.362,158.371
C02436=1037.884,318.696,-121.242,171.914,43.364,158.371
C02437=1037.890,318.943,-121.277,171.919,43.366,158.372
C02438=1037.898,319.191,-121.311,171.923,43.368,158.373
C02439=1037.904,319.438,-121.346,171.928,43.369,158.374
C02440=1037.915,319.804,-121.396,171.934,43.373,158.375
C02441=1037.926,320.170,-121.447,171.941,43.376,158.376
C02442=1037.936,320.537,-121.499,171.948,43.379,158.378
C02443=1037.947,320.903,-121.550,171.955,43.381,158.379
C02444=1037.953,321.151,-121.585,171.959,43.383,158.379
C02445=1037.961,321.398,-121.619,171.964,43.386,158.380
C02446=1037.967,321.646,-121.654,171.969,43.387,158.381
C02447=1037.975,321.893,-121.689,171.973,43.389,158.382
C02448=1037.982,322.141,-121.724,171.978,43.391,158.383
C02449=1037.989,322.389,-121.758,171.982,43.393,158.384
C02450=1037.996,322.636,-121.793,171.987,43.395,158.385
C02451=1038.004,322.883,-121.828,171.991,43.397,158.385
C02452=1038.010,323.130,-121.863,171.996,43.400,158.386
C02453=1038.019,323.378,-121.898,172.001,43.401,158.387
C02454=1038.025,323.625,-121.933,172.005,43.403,158.388
C02455=1038.033,323.872,-121.968,172.010,43.405,158.389
C02456=1038.039,324.120,-122.002,172.015,43.407,158.389
C02457=1038.047,324.368,-122.037,172.019,43.410,158.390
C02458=1038.054,324.616,-122.072,172.024,43.411,158.391
C02459=1038.062,324.863,-122.107,172.028,43.414,158.392
C02460=1038.068,325.110,-122.142,172.033,43.415,158.393
C02461=1038.077,325.358,-122.177,172.038,43.418,158.394
C02462=1038.083,325.605,-122.212,172.042,43.420,158.395
C02463=1038.091,325.852,-122.246,172.047,43.422,158.395
C02464=1038.098,326.100,-122.282,172.052,43.424,158.396
C02465=1038.105,326.348,-122.317,172.056,43.426,158.397
C02466=1038.113,326.595,-122.351,172.062,43.428,158.398
C02467=1038.120,326.842,-122.388,172.066,43.430,158.399
C02468=1038.128,327.089,-122.422,172.072,43.432,158.400
C02469=1038.135,327.337,-122.458,172.076,43.435,158.401
C02470=1038.143,327.584,-122.492,172.081,43.436,158.402
C02471=1038.149,327.832,-122.527,172.086,43.439,158.402
C02472=1038.157,328.079,-122.562,172.090,43.440,158.403
C02473=1038.164,328.327,-122.597,172.095,43.443,158.404
C02474=1038.172,328.574,-122.634,172.100,43.445,158.405
C02475=1038.179,328.821,-122.668,172.104,43.447,158.406
C02476=1038.187,329.069,-122.704,172.109,43.449,158.407
C02477=1038.194,329.316,-122.739,172.114,43.451,158.408
C02478=1038.201,329.563,-122.775,172.119,43.454,158.409
C02479=1038.208,329.811,-122.811,172.124,43.456,158.410
C02480=1038.215,330.058,-122.846,172.129,43.458,158.411
C02481=1038.223,330.306,-122.882,172.134,43.461,158.411
C02482=1038.229,330.553,-122.917,172.138,43.463,158.412
C02483=1038.237,330.801,-122.954,172.143,43.465,158.413
C02484=1038.244,331.048,-122.989,172.148,43.467,158.414
C02485=1038.251,331.295,-123.025,172.154,43.470,158.415
C02486=1038.258,331.543,-123.060,172.157,43.472,158.416
C02487=1038.265,331.789,-123.096,172.163,43.474,158.417
C02488=1038.273,332.037,-123.131,172.168,43.476,158.418
C02489=1038.280,332.284,-123.167,172.173,43.478,158.419
C02490=1038.288,332.532,-123.203,172.177,43.481,158.420
C02491=1038.295,332.780,-123.239,172.182,43.483,158.421
C02492=1038.302,333.026,-123.275,172.188,43.486,158.422
C02493=1038.310,333.274,-123.311,172.193,43.488,158.423
C02494=1038.316,333.521,-123.346,172.197,43.491,158.424
C02495=1038.324,333.769,-123.382,172.202,43.493,158.425
C02496=1038.335,334.130,-123.435,172.210,43.496,158.426
C02497=1038.346,334.492,-123.487,172.217,43.500,158.427
C02498=1038.357,334.853,-123.540,172.224,43.503,158.429
C02499=1038.367,335.215,-123.592,172.232,43.507,158.430
C02500=1038.375,335.462,-123.629,172.236,43.509,158.431
C02501=1038.382,335.709,-123.665,172.241,43.511,158.432
C02502=1038.389,335.957,-123.701,172.247,43.513,158.433
C02503=1038.397,336.204,-123.737,172.252,43.516,158.434
C02504=1038.403,336.451,-123.773,172.257,43.519,158.435
C02505=1038.411,336.699,-123.810,172.262,43.521,158.436
C02506=1038.419,336.946,-123.846,172.267,43.524,158.437
C02507=1038.426,337.193,-123.882,172.272,43.526,158.438
C02508=1038.433,337.440,-123.919,172.277,43.528,158.439
C02509=1038.440,337.688,-123.955,172.282,43.531,158.440
C02510=1038.447,337.935,-123.991,172.288,43.533,158.441
C02511=1038.455,338.182,-124.027,172.293,43.536,158.442
C02512=1038.462,338.429,-124.064,172.298,43.538,158.443
C02513=1038.470,338.677,-124.101,172.302,43.541,158.444
C02514=1038.477,338.923,-124.136,172.308,43.544,158.445
C02515=1038.485,339.171,-124.173,172.313,43.546,158.446
C02516=1038.492,339.419,-124.209,172.318,43.548,158.447
C02517=1038.500,339.665,-124.246,172.323,43.551,158.448
C02518=1038.507,339.913,-124.283,172.329,43.553,158.449
C02519=1038.514,340.160,-124.318,172.334,43.556,158.450
C02520=1038.521,340.407,-124.355,172.339,43.558,158.451
C02521=1038.529,340.654,-124.392,172.345,43.561,158.452
C02522=1038.537,340.902,-124.428,172.350,43.563,158.453
C02523=1038.545,341.149,-124.465,172.355,43.566,158.454
C02524=1038.552,341.396,-124.502,172.361,43.569,158.456
C02525=1038.560,341.644,-124.538,172.366,43.571,158.456
C02526=1038.566,341.890,-124.576,172.371,43.574,158.458
C02527=1038.574,342.138,-124.612,172.376,43.577,158.459
C02528=1038.581,342.385,-124.649,172.381,43.579,158.460
C02529=1038.589,342.632,-124.685,172.386,43.582,158.461
C02530=1038.596,342.879,-124.723,172.391,43.585,158.462
C02531=1038.604,343.126,-124.760,172.397,43.587,158.463
C02532=1038.611,343.374,-124.797,172.402,43.590,158.464
C02533=1038.619,343.621,-124.834,172.407,43.593,158.465
C02534=1038.626,343.868,-124.870,172.413,43.596,158.466
C02535=1038.634,344.115,-124.907,172.418,43.598,158.467
C02536=1038.641,344.362,-124.945,172.423,43.601,158.468
C02537=1038.649,344.610,-124.981,172.429,43.604,158.469
C02538=1038.656,344.857,-125.019,172.434,43.606,158.470
C02539=1038.664,345.104,-125.056,172.440,43.609,158.472
C02540=1038.671,345.351,-125.093,172.445,43.612,158.473
C02541=1038.679,345.598,-125.130,172.450,43.615,158.474
C02542=1038.686,345.846,-125.167,172.456,43.618,158.475
C02543=1038.694,346.093,-125.204,172.461,43.620,158.476
C02544=1038.701,346.339,-125.241,172.467,43.623,158.477
C02545=1038.709,346.587,-125.279,172.473,43.625,158.478
C02546=1038.716,346.834,-125.316,172.478,43.628,158.479
C02547=1038.724,347.081,-125.353,172.484,43.631,158.480
C02548=1038.731,347.328,-125.391,172.489,43.634,158.482
C02549=1038.739,347.575,-125.428,172.494,43.637,158.483
C02550=1038.746,347.822,-125.465,172.500,43.639,158.484
C02551=1038.754,348.069,-125.503,172.506,43.643,158.485
C02552=1038.765,348.428,-125.557,172.513,43.646,158.487
C02553=1038.776,348.785,-125.611,172.522,43.651,158.488
C02554=1038.787,349.143,-125.665,172.530,43.655,158.490
C02555=1038.799,349.501,-125.720,172.538,43.659,158.492
C02556=1038.806,349.748,-125.757,172.543,43.662,158.493
C02557=1038.813,349.995,-125.795,172.549,43.665,158.494
C02558=1038.821,350.242,-125.833,172.554,43.668,158.495
C02559=1038.829,350.489,-125.870,172.560,43.671,158.496
C02560=1038.837,350.737,-125.908,172.566,43.673,158.497
C02561=1038.844,350.983,-125.946,172.572,43.677,158.499
C02562=1038.851,351.230,-125.983,172.577,43.680,158.500
C02563=1038.859,351.477,-126.022,172.583,43.682,158.501
C02564=1038.867,351.725,-126.060,172.588,43.686,158.502
C02565=1038.874,351.972,-126.097,172.594,43.689,158.503
C02566=1038.882,352.218,-126.135,172.600,43.692,158.505
C02567=1038.889,352.465,-126.172,172.606,43.695,158.506
C02568=1038.898,352.712,-126.211,172.611,43.697,158.507
C02569=1038.905,352.960,-126.248,172.617,43.701,158.508
C02570=1038.912,353.206,-126.287,172.622,43.703,158.509
C02571=1038.920,353.454,-126.325,172.629,43.707,158.511
C02572=1038.928,353.700,-126.363,172.634,43.709,158.512
C02573=1038.935,353.947,-126.401,172.640,43.713,158.513
C02574=1038.943,354.195,-126.439,172.645,43.716,158.514
C02575=1038.951,354.441,-126.477,172.652,43.719,158.516
C02576=1038.959,354.688,-126.515,172.658,43.722,158.517
C02577=1038.967,354.935,-126.553,172.663,43.725,158.518
C02578=1038.974,355.182,-126.591,172.669,43.728,158.519
C02579=1038.983,355.429,-126.630,172.675,43.731,158.520
C02580=1038.990,355.676,-126.667,172.681,43.734,158.522
C02581=1038.998,355.923,-126.706,172.686,43.738,158.523
C02582=1039.006,356.170,-126.744,172.693,43.740,158.524
C02583=1039.014,356.417,-126.783,172.699,43.744,158.525
C02584=1039.021,356.664,-126.821,172.704,43.747,158.527
C02585=1039.029,356.911,-126.859,172.710,43.750,158.528
C02586=1039.037,357.157,-126.898,172.717,43.753,158.529
C02587=1039.045,357.405,-126.936,172.722,43.756,158.530
C02588=1039.053,357.651,-126.975,172.728,43.760,158.532
C02589=1039.061,357.898,-127.013,172.734,43.763,158.533
C02590=1039.068,358.145,-127.051,172.740,43.766,158.534
C02591=1039.076,358.392,-127.091,172.746,43.770,158.536
C02592=1039.083,358.639,-127.129,172.752,43.773,158.537
C02593=1039.091,358.886,-127.167,172.758,43.776,158.538
C02594=1039.099,359.133,-127.206,172.765,43.779,158.540
C02595=1039.107,359.380,-127.244,172.770,43.783,158.541
C02596=1039.115,359.627,-127.283,172.776,43.786,158.542
C02597=1039.123,359.873,-127.322,172.783,43.789,158.544
C02598=1039.131,360.120,-127.360,172.788,43.792,158.545
C02599=1039.138,360.367,-127.399,172.794,43.796,158.546
C02600=1039.146,360.614,-127.438,172.801,43.799,158.547
C02601=1039.155,360.861,-127.477,172.806,43.802,158.549
C02602=1039.162,361.107,-127.515,172.813,43.805,158.550
C02603=1039.170,361.355,-127.554,172.819,43.809,158.552
C02604=1039.178,361.601,-127.594,172.826,43.812,158.553
C02605=1039.186,361.849,-127.633,172.831,43.816,158.554
C02606=1039.194,362.095,-127.672,172.838,43.819,158.556
C02607=1039.202,362.342,-127.710,172.844,43.822,158.557
C02608=1039.214,362.705,-127.768,172.853,43.827,158.559
C02609=1039.225,363.070,-127.826,172.862,43.833,158.561
C02610=1039.237,363.435,-127.884,172.872,43.838,158.563
C02611=1039.248,363.798,-127.942,172.880,43.843,158.565
C02612=1039.256,364.045,-127.981,172.887,43.846,158.566
C02613=1039.265,364.292,-128.020,172.893,43.850,158.568
C02614=1039.272,364.538,-128.059,172.899,43.853,158.569
C02615=1039.280,364.785,-128.099,172.905,43.857,158.571
C02616=1039.288,365.032,-128.139,172.912,43.861,158.572
C02617=1039.296,365.278,-128.178,172.918,43.864,158.573
C02618=1039.304,365.526,-128.217,172.925,43.868,158.575
C02619=1039.312,365.772,-128.257,172.931,43.871,158.576
C02620=1039.320,366.019,-128.297,172.937,43.875,158.578
C02621=1039.328,366.265,-128.335,172.944,43.878,158.579
C02622=1039.336,366.512,-128.375,172.950,43.882,158.581
C02623=1039.344,366.759,-128.415,172.957,43.886,158.582
C02624=1039.352,367.005,-128.454,172.963,43.890,158.584
C02625=1039.360,367.252,-128.494,172.970,43.893,158.585
C02626=1039.369,367.499,-128.533,172.977,43.897,158.586
C02627=1039.376,367.746,-128.573,172.982,43.900,158.588
C02628=1039.385,367.992,-128.613,172.989,43.904,158.589
C02629=1039.393,368.239,-128.652,172.995,43.907,158.591
C02630=1039.401,368.486,-128.692,173.002,43.911,158.592
C02631=1039.409,368.732,-128.732,173.009,43.915,158.594
C02632=1039.417,368.979,-128.772,173.015,43.919,158.595
C02633=1039.425,369.226,-128.812,173.022,43.922,158.597
C02634=1039.434,369.472,-128.851,173.029,43.926,158.598
C02635=1039.441,369.719,-128.891,173.035,43.930,158.600
C02636=1039.451,369.966,-128.931,173.042,43.934,158.601
C02637=1039.458,370.213,-128.971,173.048,43.937,158.603
C02638=1039.467,370.459,-129.011,173.054,43.941,158.604
C02639=1039.475,370.706,-129.051,173.061,43.945,158.606
C02640=1039.483,370.953,-129.091,173.068,43.949,158.607
C02641=1039.491,371.199,-129.132,173.075,43.952,158.609
C02642=1039.499,371.445,-129.171,173.081,43.956,158.610
C02643=1039.507,371.692,-129.212,173.088,43.960,158.612
C02644=1039.515,371.939,-129.252,173.095,43.964,158.613
C02645=1039.523,372.186,-129.293,173.101,43.968,158.615
C02646=1039.532,372.432,-129.333,173.108,43.972,158.616
C02647=1039.540,372.678,-129.373,173.115,43.976,158.618
C02648=1039.548,372.925,-129.413,173.122,43.980,158.620
C02649=1039.556,373.171,-129.454,173.128,43.984,158.621
C02650=1039.564,373.419,-129.494,173.135,43.988,158.623
C02651=1039.572,373.665,-129.535,173.142,43.992,158.624
C02652=1039.581,373.911,-129.575,173.149,43.995,158.626
C02653=1039.589,374.157,-129.615,173.157,43.999,158.627
C02654=1039.598,374.404,-129.656,173.163,44.003,158.629
C02655=1039.606,374.650,-129.697,173.170,44.008,158.631
C02656=1039.614,374.897,-129.737,173.177,44.011,158.632
C02657=1039.622,375.144,-129.778,173.184,44.015,158.634
C02658=1039.631,375.390,-129.818,173.191,44.019,158.635
C02659=1039.639,375.637,-129.859,173.198,44.023,158.637
C02660=1039.648,375.884,-129.900,173.205,44.028,158.639
C02661=1039.656,376.130,-129.940,173.211,44.031,158.640
C02662=1039.664,376.377,-129.981,173.218,44.036,158.642
C02663=1039.672,376.623,-130.022,173.226,44.040,158.644
C02664=1039.686,377.007,-130.086,173.237,44.046,158.646
C02665=1039.699,377.390,-130.149,173.248,44.052,158.649
C02666=1039.712,377.775,-130.213,173.259,44.059,158.651
C02667=1039.726,378.159,-130.277,173.270,44.065,158.654
C02668=1039.734,378.406,-130.318,173.277,44.069,158.655
C02669=1039.743,378.653,-130.359,173.284,44.074,158.657
C02670=1039.751,378.898,-130.400,173.291,44.078,158.659
C02671=1039.760,379.145,-130.441,173.299,44.082,158.661
C02672=1039.768,379.391,-130.482,173.306,44.086,158.662
C02673=1039.776,379.638,-130.524,173.313,44.090,158.664
C02674=1039.784,379.884,-130.565,173.320,44.095,158.666
C02675=1039.793,380.131,-130.606,173.328,44.099,158.668
C02676=1039.801,380.376,-130.648,173.335,44.104,158.669
C02677=1039.810,380.623,-130.689,173.342,44.108,158.671
C02678=1039.819,380.870,-130.730,173.349,44.112,158.673
C02679=1039.826,381.116,-130.772,173.357,44.117,158.674
C02680=1039.835,381.362,-130.814,173.364,44.121,158.676
C02681=1039.844,381.609,-130.855,173.371,44.125,158.678
C02682=1039.852,381.855,-130.896,173.378,44.129,158.680
C02683=1039.861,382.101,-130.938,173.386,44.134,158.681
C02684=1039.869,382.348,-130.980,173.393,44.138,158.683
C02685=1039.878,382.593,-131.022,173.401,44.143,158.685
C02686=1039.887,382.840,-131.063,173.408,44.147,158.687
C02687=1039.895,383.087,-131.104,173.416,44.152,158.689
C02688=1039.904,383.333,-131.146,173.424,44.156,158.690
C02689=1039.912,383.579,-131.188,173.431,44.161,158.692
C02690=1039.921,383.826,-131.230,173.438,44.165,158.694
C02691=1039.930,384.072,-131.271,173.446,44.170,158.696
C02692=1039.938,384.318,-131.313,173.453,44.174,158.698
C02693=1039.948,384.564,-131.356,173.460,44.179,158.699
C02694=1039.956,384.811,-131.398,173.469,44.183,158.701
C02695=1039.964,385.056,-131.439,173.476,44.188,158.703
C02696=1039.973,385.303,-131.481,173.484,44.192,158.705
C02697=1039.982,385.549,-131.523,173.491,44.197,158.707
C02698=1039.990,385.796,-131.565,173.500,44.202,158.709
C02699=1040.000,386.041,-131.607,173.507,44.206,158.710
C02700=1040.008,386.288,-131.649,173.514,44.211,158.712
C02701=1040.017,386.534,-131.691,173.522,44.215,158.714
C02702=1040.027,386.780,-131.733,173.530,44.220,158.716
C02703=1040.035,387.027,-131.776,173.538,44.225,158.718
C02704=1040.044,387.273,-131.817,173.545,44.229,158.720
C02705=1040.053,387.519,-131.860,173.554,44.234,158.722
C02706=1040.062,387.765,-131.901,173.561,44.239,158.724
C02707=1040.070,388.011,-131.944,173.569,44.243,158.725
C02708=1040.079,388.258,-131.986,173.577,44.248,158.727
C02709=1040.088,388.504,-132.029,173.585,44.253,158.729
C02710=1040.097,388.749,-132.072,173.592,44.257,158.731
C02711=1040.105,388.996,-132.114,173.601,44.262,158.733
C02712=1040.115,389.242,-132.157,173.608,44.267,158.735
C02713=1040.124,389.489,-132.200,173.616,44.272,158.737
C02714=1040.133,389.734,-132.242,173.625,44.277,158.739
C02715=1040.141,389.981,-132.285,173.632,44.282,158.741
C02716=1040.150,390.227,-132.327,173.640,44.286,158.743
C02717=1040.159,390.473,-132.370,173.648,44.291,158.745
C02718=1040.168,390.718,-132.412,173.656,44.296,158.747
C02719=1040.177,390.965,-132.456,173.665,44.301,158.749
C02720=1040.184,391.174,-132.492,173.671,44.306,158.751
C02721=1040.192,391.383,-132.528,173.678,44.310,158.752
C02722=1040.200,391.592,-132.565,173.685,44.314,158.754
C02723=1040.208,391.801,-132.602,173.692,44.318,158.756
C02724=1040.215,392.010,-132.638,173.699,44.322,158.758
C02725=1040.223,392.219,-132.674,173.706,44.326,158.759
C02726=1040.231,392.428,-132.711,173.712,44.331,158.761
C02727=1040.238,392.638,-132.748,173.720,44.335,158.763
C02728=1040.247,392.884,-132.790,173.729,44.340,158.765
C02729=1040.257,393.130,-132.834,173.736,44.345,158.767
C02730=1040.265,393.376,-132.877,173.745,44.350,158.769
C02731=1040.274,393.622,-132.920,173.753,44.355,158.771
C02732=1040.283,393.868,-132.963,173.761,44.360,158.773
C02733=1040.292,394.114,-133.007,173.769,44.365,158.775
C02734=1040.302,394.360,-133.050,173.778,44.370,158.777
C02735=1040.311,394.606,-133.094,173.787,44.375,158.779
C02736=1040.320,394.852,-133.137,173.794,44.381,158.781
C02737=1040.329,395.098,-133.180,173.803,44.386,158.783
C02738=1040.339,395.344,-133.223,173.811,44.391,158.786
C02739=1040.347,395.590,-133.267,173.820,44.396,158.788
C02740=1040.356,395.835,-133.311,173.829,44.402,158.790
C02741=1040.365,396.082,-133.354,173.837,44.407,158.792
C02742=1040.375,396.328,-133.398,173.845,44.412,158.794
C02743=1040.384,396.573,-133.442,173.854,44.417,158.796
C02744=1040.394,396.819,-133.486,173.862,44.423,158.798
C02745=1040.402,397.065,-133.529,173.871,44.428,158.801
C02746=1040.412,397.311,-133.573,173.880,44.433,158.803
C02747=1040.420,397.557,-133.617,173.889,44.438,158.805
C02748=1040.430,397.803,-133.661,173.897,44.444,158.807
C02749=1040.439,398.049,-133.705,173.906,44.449,158.809
C02750=1040.449,398.294,-133.748,173.915,44.455,158.812
C02751=1040.458,398.540,-133.792,173.924,44.460,158.814
C02752=1040.468,398.787,-133.836,173.932,44.465,158.816
C02753=1040.476,399.032,-133.880,173.941,44.471,158.818
C02754=1040.486,399.278,-133.924,173.950,44.477,158.821
C02755=1040.495,399.524,-133.969,173.959,44.482,158.823
C02756=1040.505,399.770,-134.013,173.968,44.487,158.825
C02757=1040.514,400.016,-134.057,173.977,44.493,158.827
C02758=1040.523,400.261,-134.101,173.985,44.498,158.830
C02759=1040.533,400.507,-134.146,173.994,44.504,158.832
C02760=1040.542,400.753,-134.190,174.003,44.510,158.834
C02761=1040.552,400.999,-134.234,174.012,44.515,158.836
C02762=1040.561,401.245,-134.279,174.021,44.521,158.839
C02763=1040.571,401.491,-134.323,174.030,44.526,158.841
C02764=1040.580,401.736,-134.368,174.039,44.532,158.843
C02765=1040.590,401.982,-134.412,174.048,44.537,158.846
C02766=1040.600,402.228,-134.457,174.057,44.543,158.848
C02767=1040.608,402.474,-134.501,174.067,44.549,158.850
C02768=1040.618,402.720,-134.546,174.076,44.554,158.853
C02769=1040.628,402.965,-134.591,174.085,44.560,158.855
C02770=1040.637,403.212,-134.635,174.094,44.566,158.858
C02771=1040.647,403.457,-134.680,174.103,44.572,158.860
C02772=1040.657,403.703,-134.725,174.113,44.578,158.862
C02773=1040.666,403.948,-134.770,174.122,44.583,158.865
C02774=1040.675,404.194,-134.815,174.131,44.589,158.867
C02775=1040.685,404.439,-134.860,174.140,44.595,158.869
C02776=1040.694,404.685,-134.905,174.150,44.601,158.872
C02777=1040.704,404.931,-134.950,174.159,44.607,158.874
C02778=1040.714,405.177,-134.995,174.168,44.612,158.877
C02779=1040.723,405.423,-135.041,174.177,44.618,158.879
C02780=1040.732,405.642,-135.080,174.186,44.624,158.882
C02781=1040.740,405.860,-135.121,174.194,44.629,158.884
C02782=1040.749,406.080,-135.161,174.203,44.635,158.886
C02783=1040.757,406.299,-135.201,174.211,44.640,158.888
C02784=1040.767,406.517,-135.242,174.220,44.645,158.890
C02785=1040.775,406.736,-135.283,174.228,44.650,158.893
C02786=1040.783,406.955,-135.323,174.237,44.656,158.895
C02787=1040.792,407.174,-135.363,174.246,44.661,158.897
C02788=1040.802,407.420,-135.409,174.256,44.667,158.900
C02789=1040.811,407.666,-135.454,174.265,44.673,158.902
C02790=1040.821,407.911,-135.499,174.275,44.679,158.905
C02791=1040.832,408.157,-135.545,174.285,44.685,158.907
C02792=1040.841,408.402,-135.591,174.294,44.691,158.910
C02793=1040.851,408.648,-135.637,174.304,44.698,158.912
C02794=1040.861,408.893,-135.682,174.314,44.704,158.915
C02795=1040.871,409.139,-135.728,174.324,44.710,158.918
C02796=1040.881,409.384,-135.773,174.333,44.716,158.920
C02797=1040.891,409.630,-135.820,174.344,44.722,158.923
C02798=1040.901,409.877,-135.865,174.353,44.729,158.925
C02799=1040.911,410.121,-135.911,174.364,44.735,158.928
C02800=1040.921,410.367,-135.957,174.373,44.741,158.931
C02801=1040.931,410.612,-136.003,174.383,44.747,158.933
C02802=1040.942,410.858,-136.049,174.394,44.754,158.936
C02803=1040.952,411.104,-136.095,174.403,44.760,158.939
C02804=1040.962,411.349,-136.141,174.414,44.766,158.941
C02805=1040.971,411.594,-136.187,174.424,44.773,158.944
C02806=1040.982,411.840,-136.233,174.434,44.779,158.947
C02807=1040.992,412.086,-136.280,174.445,44.785,158.949
C02808=1041.002,412.332,-136.326,174.455,44.792,158.952
C02809=1041.012,412.577,-136.372,174.465,44.798,158.955
C02810=1041.022,412.822,-136.419,174.475,44.805,158.958
C02811=1041.032,413.068,-136.465,174.486,44.811,158.960
C02812=1041.043,413.314,-136.511,174.496,44.818,158.963
C02813=1041.053,413.559,-136.558,174.506,44.824,158.966
C02814=1041.063,413.805,-136.605,174.517,44.831,158.969
C02815=1041.072,414.049,-136.652,174.527,44.838,158.972
C02816=1041.083,414.295,-136.698,174.538,44.844,158.974
C02817=1041.093,414.540,-136.745,174.549,44.851,158.977
C02818=1041.103,414.786,-136.791,174.559,44.857,158.980
C02819=1041.114,415.031,-136.838,174.569,44.864,158.983
C02820=1041.124,415.276,-136.885,174.580,44.870,158.986
C02821=1041.134,415.522,-136.932,174.591,44.877,158.988
C02822=1041.144,415.768,-136.979,174.602,44.884,158.991
C02823=1041.155,416.013,-137.026,174.612,44.891,158.994
C02824=1041.165,416.258,-137.073,174.623,44.897,158.997
C02825=1041.176,416.504,-137.120,174.634,44.904,159.000
C02826=1041.186,416.749,-137.168,174.645,44.911,159.003
C02827=1041.197,416.994,-137.214,174.656,44.918,159.006
C02828=1041.207,417.239,-137.261,174.667,44.925,159.009
C02829=1041.218,417.485,-137.309,174.678,44.931,159.012
C02830=1041.228,417.730,-137.356,174.689,44.938,159.015
C02831=1041.239,417.976,-137.403,174.700,44.945,159.018
C02832=1041.249,418.221,-137.450,174.711,44.952,159.021
C02833=1041.260,418.466,-137.498,174.722,44.959,159.024
C02834=1041.270,418.711,-137.545,174.733,44.966,159.027
C02835=1041.281,418.957,-137.593,174.744,44.973,159.030
C02836=1041.291,419.201,-137.641,174.755,44.980,159.033
C02837=1041.302,419.447,-137.688,174.766,44.987,159.036
C02838=1041.313,419.692,-137.736,174.778,44.995,159.039
C02839=1041.323,419.937,-137.783,174.789,45.001,159.042
C02840=1041.336,420.237,-137.842,174.803,45.010,159.046
C02841=1041.349,420.537,-137.901,174.816,45.019,159.049
C02842=1041.362,420.837,-137.960,174.830,45.028,159.053
C02843=1041.375,421.137,-138.018,174.845,45.037,159.057
C02844=1041.385,421.382,-138.066,174.856,45.044,159.060
C02845=1041.396,421.627,-138.114,174.867,45.051,159.063
C02846=1041.408,421.872,-138.163,174.880,45.058,159.067
C02847=1041.418,422.117,-138.210,174.891,45.066,159.070
C02848=1041.435,422.508,-138.288,174.910,45.077,159.075
C02849=1041.453,422.899,-138.365,174.928,45.089,159.080
C02850=1041.470,423.291,-138.442,174.947,45.101,159.085
C02851=1041.488,423.682,-138.519,174.966,45.112,159.090
C02852=1041.499,423.928,-138.567,174.978,45.120,159.094
C02853=1041.510,424.172,-138.616,174.990,45.127,159.097
C02854=1041.521,424.417,-138.664,175.001,45.135,159.100
C02855=1041.531,424.663,-138.713,175.014,45.142,159.103
C02856=1041.543,424.908,-138.762,175.026,45.150,159.107
C02857=1041.554,425.152,-138.811,175.038,45.158,159.110
C02858=1041.564,425.398,-138.860,175.050,45.165,159.113
C02859=1041.575,425.642,-138.909,175.062,45.172,159.117
C02860=1041.587,425.887,-138.958,175.075,45.180,159.120
C02861=1041.598,426.132,-139.006,175.087,45.188,159.124
C02862=1041.608,426.377,-139.056,175.099,45.196,159.127
C02863=1041.620,426.622,-139.105,175.112,45.203,159.130
C02864=1041.631,426.867,-139.154,175.124,45.211,159.134
C02865=1041.642,427.112,-139.203,175.137,45.219,159.137
C02866=1041.653,427.356,-139.252,175.149,45.226,159.141
C02867=1041.665,427.601,-139.301,175.161,45.235,159.144
C02868=1041.677,427.847,-139.351,175.174,45.242,159.148
C02869=1041.687,428.092,-139.400,175.187,45.250,159.151
C02870=1041.699,428.336,-139.449,175.200,45.258,159.155
C02871=1041.710,428.581,-139.500,175.212,45.266,159.158
C02872=1041.722,428.826,-139.549,175.225,45.274,159.162
C02873=1041.732,429.071,-139.599,175.237,45.282,159.165
C02874=1041.744,429.315,-139.648,175.250,45.290,159.169
C02875=1041.755,429.561,-139.698,175.263,45.298,159.172
C02876=1041.767,429.805,-139.748,175.276,45.306,159.176
C02877=1041.778,430.050,-139.798,175.289,45.314,159.180
C02878=1041.789,430.294,-139.847,175.302,45.322,159.183
C02879=1041.800,430.539,-139.898,175.315,45.330,159.187
C02880=1041.813,430.784,-139.948,175.328,45.338,159.191
C02881=1041.823,431.029,-139.997,175.342,45.347,159.194
C02882=1041.835,431.274,-140.048,175.356,45.354,159.198
C02883=1041.847,431.518,-140.098,175.369,45.363,159.202
C02884=1041.858,431.763,-140.148,175.382,45.371,159.205
C02885=1041.870,432.007,-140.198,175.395,45.379,159.209
C02886=1041.882,432.252,-140.249,175.408,45.388,159.213
C02887=1041.893,432.497,-140.299,175.422,45.396,159.217
C02888=1041.905,432.742,-140.349,175.436,45.404,159.221
C02889=1041.917,432.986,-140.400,175.449,45.413,159.224
C02890=1041.928,433.230,-140.450,175.462,45.421,159.228
C02891=1041.941,433.475,-140.500,175.477,45.429,159.232
C02892=1041.953,433.720,-140.552,175.490,45.438,159.236
C02893=1041.964,433.964,-140.602,175.503,45.446,159.240
C02894=1041.976,434.209,-140.652,175.518,45.454,159.243
C02895=1041.988,434.453,-140.704,175.531,45.463,159.247
C02896=1041.999,434.684,-140.752,175.544,45.471,159.251
C02897=1042.011,434.916,-140.799,175.558,45.480,159.255
C02898=1042.022,435.147,-140.847,175.572,45.487,159.259
C02899=1042.033,435.378,-140.896,175.585,45.496,159.262
C02900=1042.045,435.610,-140.944,175.598,45.503,159.266
C02901=1042.056,435.842,-140.993,175.611,45.512,159.270
C02902=1042.068,436.073,-141.041,175.625,45.520,159.274
C02903=1042.079,436.304,-141.089,175.638,45.529,159.277
C02904=1042.091,436.548,-141.141,175.652,45.537,159.281
C02905=1042.103,436.793,-141.192,175.667,45.546,159.285
C02906=1042.115,437.037,-141.244,175.681,45.555,159.290
C02907=1042.127,437.281,-141.296,175.695,45.563,159.294
C02908=1042.140,437.525,-141.346,175.710,45.573,159.298
C02909=1042.152,437.770,-141.398,175.725,45.581,159.302
C02910=1042.163,438.014,-141.449,175.740,45.590,159.306
C02911=1042.176,438.259,-141.502,175.754,45.599,159.310
C02912=1042.188,438.503,-141.553,175.768,45.608,159.314
C02913=1042.200,438.747,-141.605,175.783,45.617,159.319
C02914=1042.212,438.991,-141.657,175.798,45.626,159.323
C02915=1042.225,439.235,-141.708,175.813,45.635,159.327
C02916=1042.238,439.480,-141.761,175.828,45.644,159.331
C02917=1042.250,439.724,-141.813,175.843,45.653,159.335
C02918=1042.263,439.968,-141.865,175.858,45.662,159.340
C02919=1042.275,440.212,-141.917,175.874,45.672,159.344
C02920=1042.287,440.456,-141.970,175.889,45.681,159.348
C02921=1042.300,440.701,-142.022,175.904,45.690,159.353
C02922=1042.312,440.945,-142.074,175.919,45.699,159.357
C02923=1042.325,441.189,-142.127,175.934,45.708,159.361
C02924=1042.337,441.433,-142.179,175.951,45.718,159.366
C02925=1042.350,441.678,-142.231,175.966,45.727,159.370
C02926=1042.363,441.922,-142.284,175.981,45.736,159.375
C02927=1042.375,442.166,-142.337,175.997,45.746,159.379
C02928=1042.388,442.410,-142.390,176.012,45.755,159.384
C02929=1042.401,442.654,-142.442,176.028,45.765,159.388
C02930=1042.414,442.897,-142.495,176.044,45.775,159.393
C02931=1042.426,443.142,-142.548,176.060,45.784,159.397
C02932=1042.440,443.386,-142.601,176.076,45.793,159.402
C02933=1042.453,443.630,-142.654,176.091,45.803,159.406
C02934=1042.465,443.873,-142.707,176.108,45.813,159.411
C02935=1042.478,444.117,-142.760,176.124,45.822,159.416
C02936=1042.491,444.361,-142.813,176.140,45.832,159.420
C02937=1042.504,444.604,-142.866,176.156,45.842,159.425
C02938=1042.517,444.848,-142.919,176.173,45.851,159.429
C02939=1042.530,445.092,-142.972,176.188,45.861,159.434
C02940=1042.544,445.334,-143.025,176.205,45.870,159.439
C02941=1042.559,445.578,-143.077,176.221,45.880,159.443
C02942=1042.573,445.822,-143.128,176.238,45.889,159.448
C02943=1042.589,446.065,-143.180,176.255,45.898,159.453
C02944=1042.606,446.309,-143.230,176.272,45.907,159.457
C02945=1042.622,446.553,-143.280,176.288,45.916,159.462
C02946=1042.640,446.797,-143.330,176.306,45.925,159.466
C02947=1042.658,447.041,-143.379,176.323,45.934,159.471
C02948=1042.677,447.285,-143.428,176.340,45.942,159.475
C02949=1042.696,447.530,-143.476,176.356,45.951,159.480
C02950=1042.716,447.774,-143.524,176.374,45.959,159.484
C02951=1042.737,448.018,-143.571,176.391,45.967,159.489
C02952=1042.758,448.263,-143.618,176.408,45.976,159.493
C02953=1042.780,448.508,-143.664,176.426,45.984,159.497
C02954=1042.802,448.752,-143.709,176.444,45.992,159.502
C02955=1042.824,448.998,-143.755,176.461,46.000,159.506
C02956=1042.858,449.347,-143.819,176.486,46.011,159.513
C02957=1042.893,449.695,-143.882,176.512,46.022,159.519
C02958=1042.929,450.044,-143.943,176.537,46.033,159.525
C02959=1042.966,450.394,-144.004,176.563,46.043,159.531
C02960=1042.993,450.640,-144.047,176.581,46.050,159.535
C02961=1043.021,450.886,-144.088,176.600,46.057,159.539
C02962=1043.049,451.131,-144.129,176.617,46.064,159.543
C02963=1043.078,451.376,-144.170,176.636,46.071,159.548
C02964=1042.777,451.417,-144.483,176.638,46.151,159.572
C02965=1042.749,451.173,-144.443,176.620,46.144,159.568
C02966=1042.720,450.927,-144.402,176.602,46.137,159.564
C02967=1042.693,450.681,-144.360,176.583,46.130,159.559
C02968=1042.665,450.436,-144.319,176.565,46.123,159.555
C02969=1042.629,450.103,-144.261,176.540,46.113,159.549
C02970=1042.595,449.769,-144.202,176.516,46.103,159.543
C02971=1042.561,449.436,-144.143,176.491,46.093,159.537
C02972=1042.529,449.102,-144.082,176.467,46.082,159.531
C02973=1042.505,448.857,-144.036,176.449,46.075,159.527
C02974=1042.482,448.612,-143.991,176.432,46.067,159.523
C02975=1042.460,448.368,-143.945,176.414,46.059,159.518
C02976=1042.439,448.123,-143.898,176.397,46.051,159.514
C02977=1042.417,447.879,-143.852,176.380,46.042,159.510
C02978=1042.398,447.634,-143.804,176.363,46.034,159.505
C02979=1042.378,447.390,-143.756,176.346,46.026,159.501
C02980=1042.359,447.146,-143.708,176.328,46.017,159.496
C02981=1042.341,446.902,-143.658,176.311,46.008,159.492
C02982=1042.323,446.657,-143.609,176.294,46.000,159.487
C02983=1042.306,446.413,-143.559,176.277,45.991,159.483
C02984=1042.288,446.170,-143.509,176.260,45.982,159.478
C02985=1042.273,445.926,-143.458,176.243,45.973,159.473
C02986=1042.257,445.683,-143.406,176.227,45.964,159.469
C02987=1042.242,445.439,-143.356,176.209,45.955,159.464
C02988=1042.228,445.196,-143.303,176.194,45.945,159.460
C02989=1042.214,444.952,-143.250,176.177,45.936,159.455
C02990=1042.201,444.709,-143.197,176.161,45.926,159.450
C02991=1042.188,444.465,-143.144,176.144,45.917,159.446
C02992=1042.175,444.223,-143.091,176.128,45.907,159.441
C02993=1042.162,443.979,-143.037,176.112,45.897,159.436
C02994=1042.149,443.735,-142.984,176.096,45.888,159.432
C02995=1042.136,443.490,-142.932,176.079,45.878,159.427
C02996=1042.124,443.247,-142.879,176.064,45.869,159.423
C02997=1042.111,443.003,-142.826,176.047,45.860,159.418
C02998=1042.098,442.759,-142.773,176.032,45.850,159.413
C02999=1042.085,442.515,-142.720,176.016,45.841,159.409
C03000=1042.072,442.271,-142.667,176.000,45.831,159.404
C03001=1042.060,442.027,-142.615,175.984,45.822,159.400
C03002=1042.046,441.783,-142.562,175.969,45.813,159.396
C03003=1042.034,441.539,-142.509,175.954,45.804,159.391
C03004=1042.021,441.294,-142.457,175.937,45.794,159.387
C03005=1042.009,441.050,-142.405,175.922,45.785,159.382
C03006=1041.996,440.806,-142.352,175.907,45.776,159.378
C03007=1041.984,440.562,-142.299,175.891,45.767,159.374
C03008=1041.971,440.318,-142.247,175.876,45.758,159.369
C03009=1041.959,440.074,-142.195,175.861,45.749,159.365
C03010=1041.946,439.829,-142.142,175.846,45.740,159.361
C03011=1041.934,439.585,-142.091,175.831,45.731,159.356
C03012=1041.921,439.341,-142.039,175.816,45.722,159.352
C03013=1041.909,439.097,-141.987,175.801,45.713,159.348
C03014=1041.896,438.853,-141.935,175.786,45.703,159.344
C03015=1041.885,438.608,-141.883,175.771,45.694,159.339
C03016=1041.872,438.364,-141.831,175.756,45.686,159.335
C03017=1041.860,438.119,-141.780,175.741,45.677,159.331
C03018=1041.848,437.875,-141.727,175.727,45.668,159.327
C03019=1041.836,437.631,-141.676,175.712,45.659,159.323
C03020=1041.823,437.387,-141.625,175.697,45.650,159.319
C03021=1041.811,437.143,-141.573,175.682,45.642,159.315
C03022=1041.799,436.898,-141.522,175.669,45.633,159.310
C03023=1041.787,436.653,-141.470,175.654,45.624,159.306
C03024=1041.774,436.409,-141.419,175.639,45.616,159.302
C03025=1041.763,436.177,-141.370,175.626,45.607,159.299
C03026=1041.752,435.945,-141.321,175.613,45.599,159.295
C03027=1041.741,435.713,-141.273,175.598,45.591,159.291
C03028=1041.728,435.481,-141.225,175.585,45.583,159.287
C03029=1041.717,435.249,-141.176,175.572,45.575,159.283
C03030=1041.706,435.016,-141.127,175.559,45.566,159.280
C03031=1041.695,434.785,-141.080,175.545,45.559,159.276
C03032=1041.683,434.553,-141.031,175.532,45.551,159.272
C03033=1041.672,434.307,-140.980,175.518,45.542,159.268
C03034=1041.659,434.063,-140.929,175.504,45.534,159.264
C03035=1041.647,433.818,-140.879,175.490,45.525,159.261
C03036=1041.635,433.575,-140.828,175.477,45.517,159.257
C03037=1041.624,433.329,-140.777,175.462,45.509,159.253
C03038=1041.612,433.085,-140.727,175.449,45.500,159.249
C03039=1041.601,432.840,-140.677,175.436,45.492,159.245
C03040=1041.588,432.596,-140.626,175.422,45.484,159.241
C03041=1041.576,432.351,-140.575,175.408,45.475,159.238
C03042=1041.565,432.107,-140.526,175.395,45.467,159.234
C03043=1041.553,431.862,-140.475,175.381,45.459,159.230
C03044=1041.541,431.618,-140.425,175.368,45.451,159.226
C03045=1041.530,431.372,-140.375,175.355,45.443,159.223
C03046=1041.519,431.128,-140.324,175.341,45.434,159.219
C03047=1041.507,430.883,-140.274,175.328,45.427,159.215
C03048=1041.496,430.639,-140.224,175.315,45.419,159.212
C03049=1041.484,430.393,-140.175,175.302,45.410,159.208
C03050=1041.473,430.149,-140.124,175.288,45.402,159.204
C03051=1041.461,429.905,-140.074,175.275,45.394,159.201
C03052=1041.450,429.659,-140.024,175.262,45.386,159.197
C03053=1041.438,429.415,-139.975,175.249,45.379,159.193
C03054=1041.427,429.170,-139.925,175.236,45.371,159.190
C03055=1041.416,428.926,-139.875,175.224,45.362,159.186
C03056=1041.404,428.680,-139.825,175.211,45.354,159.183
C03057=1041.393,428.436,-139.776,175.198,45.347,159.179
C03058=1041.382,428.191,-139.726,175.185,45.339,159.176
C03059=1041.370,427.946,-139.677,175.173,45.331,159.172
C03060=1041.359,427.701,-139.628,175.160,45.323,159.169
C03061=1041.348,427.455,-139.578,175.147,45.316,159.165
C03062=1041.336,427.211,-139.529,175.135,45.308,159.162
C03063=1041.325,426.966,-139.480,175.122,45.300,159.158
C03064=1041.314,426.721,-139.431,175.110,45.293,159.155
C03065=1041.303,426.476,-139.381,175.097,45.285,159.151
C03066=1041.292,426.231,-139.332,175.085,45.277,159.148
C03067=1041.280,425.987,-139.283,175.072,45.270,159.145
C03068=1041.270,425.741,-139.235,175.060,45.262,159.141
C03069=1041.258,425.496,-139.186,175.048,45.254,159.138
C03070=1041.247,425.252,-139.137,175.035,45.247,159.134
C03071=1041.236,425.008,-139.088,175.023,45.240,159.131
C03072=1041.226,424.762,-139.039,175.011,45.232,159.128
C03073=1041.214,424.517,-138.990,174.999,45.225,159.124
C03074=1041.203,424.272,-138.942,174.987,45.217,159.121
C03075=1041.192,424.026,-138.893,174.975,45.210,159.118
C03076=1041.181,423.782,-138.844,174.963,45.202,159.115
C03077=1041.170,423.537,-138.796,174.951,45.195,159.111
C03078=1041.159,423.292,-138.748,174.939,45.188,159.108
C03079=1041.148,423.046,-138.700,174.928,45.180,159.105
C03080=1041.137,422.801,-138.650,174.915,45.173,159.102
C03081=1041.127,422.557,-138.602,174.904,45.166,159.098
C03082=1041.116,422.311,-138.554,174.892,45.159,159.095
C03083=1041.105,422.066,-138.506,174.880,45.152,159.092
C03084=1041.094,421.821,-138.458,174.869,45.144,159.089
C03085=1041.084,421.597,-138.414,174.858,45.138,159.086
C03086=1041.074,421.373,-138.370,174.847,45.131,159.083
C03087=1041.064,421.148,-138.327,174.837,45.124,159.080
C03088=1041.055,420.925,-138.283,174.826,45.118,159.077
C03089=1041.045,420.700,-138.238,174.816,45.111,159.075
C03090=1041.035,420.477,-138.195,174.805,45.105,159.072
C03091=1041.025,420.252,-138.151,174.794,45.098,159.069
C03092=1041.015,420.028,-138.107,174.785,45.092,159.066
C03093=1041.005,419.783,-138.060,174.773,45.085,159.063
C03094=1040.994,419.538,-138.012,174.762,45.078,159.060
C03095=1040.983,419.293,-137.964,174.750,45.071,159.057
C03096=1040.973,419.048,-137.917,174.739,45.064,159.054
C03097=1040.962,418.802,-137.868,174.728,45.057,159.051
C03098=1040.952,418.557,-137.821,174.717,45.050,159.048
C03099=1040.942,418.312,-137.774,174.706,45.043,159.045
C03100=1040.930,418.066,-137.726,174.694,45.036,159.042
C03101=1040.920,417.821,-137.678,174.683,45.029,159.039
C03102=1040.910,417.576,-137.631,174.672,45.023,159.036
C03103=1040.900,417.331,-137.584,174.661,45.016,159.033
C03104=1040.889,417.085,-137.536,174.650,45.009,159.030
C03105=1040.878,416.840,-137.490,174.639,45.002,159.027
C03106=1040.868,416.594,-137.443,174.628,44.995,159.024
C03107=1040.858,416.349,-137.395,174.618,44.989,159.021
C03108=1040.848,416.104,-137.348,174.607,44.982,159.018
C03109=1040.836,415.858,-137.301,174.596,44.975,159.015
C03110=1040.826,415.612,-137.255,174.585,44.968,159.012
C03111=1040.816,415.367,-137.207,174.575,44.962,159.010
C03112=1040.805,415.122,-137.161,174.564,44.955,159.007
C03113=1040.789,414.725,-137.085,174.546,44.945,159.002
C03114=1040.772,414.327,-137.009,174.529,44.934,158.998
C03115=1040.755,413.929,-136.934,174.513,44.923,158.993
C03116=1040.740,413.532,-136.858,174.496,44.913,158.989
C03117=1040.729,413.286,-136.812,174.485,44.907,158.986
C03118=1040.719,413.041,-136.765,174.474,44.900,158.983
C03119=1040.709,412.795,-136.718,174.464,44.893,158.980
C03120=1040.699,412.549,-136.672,174.454,44.887,158.977
C03121=1040.689,412.305,-136.626,174.444,44.881,158.975
C03122=1040.679,412.059,-136.579,174.433,44.874,158.972
C03123=1040.669,411.813,-136.533,174.423,44.868,158.969
C03124=1040.658,411.567,-136.487,174.413,44.862,158.967
C03125=1040.648,411.322,-136.441,174.402,44.856,158.964
C03126=1040.639,411.077,-136.395,174.393,44.849,158.961
C03127=1040.628,410.831,-136.349,174.382,44.843,158.958
C03128=1040.618,410.585,-136.302,174.373,44.837,158.956
C03129=1040.608,410.340,-136.257,174.362,44.830,158.953
C03130=1040.597,410.095,-136.211,174.352,44.824,158.951
C03131=1040.588,409.849,-136.164,174.342,44.818,158.948
C03132=1040.578,409.603,-136.119,174.332,44.812,158.945
C03133=1040.568,409.357,-136.073,174.322,44.806,158.943
C03134=1040.558,409.112,-136.027,174.312,44.800,158.940
C03135=1040.548,408.866,-135.982,174.303,44.794,158.938
C03136=1040.538,408.621,-135.936,174.292,44.787,158.935
C03137=1040.528,408.375,-135.890,174.283,44.781,158.932
C03138=1040.518,408.130,-135.845,174.273,44.775,158.930
C03139=1040.508,407.884,-135.799,174.263,44.770,158.927
C03140=1040.498,407.638,-135.754,174.254,44.764,158.925
C03141=1040.488,407.393,-135.708,174.244,44.758,158.922
C03142=1040.479,407.147,-135.663,174.234,44.752,158.920
C03143=1040.469,406.901,-135.618,174.224,44.746,158.917
C03144=1040.458,406.656,-135.572,174.215,44.740,158.915
C03145=1040.447,406.368,-135.519,174.203,44.732,158.912
C03146=1040.436,406.081,-135.466,174.192,44.725,158.909
C03147=1040.424,405.793,-135.413,174.181,44.718,158.906
C03148=1040.413,405.505,-135.360,174.170,44.711,158.903
C03149=1040.404,405.260,-135.314,174.161,44.706,158.901
C03150=1040.394,405.014,-135.269,174.151,44.700,158.898
C03151=1040.385,404.769,-135.224,174.141,44.694,158.896
C03152=1040.376,404.523,-135.179,174.132,44.689,158.893
C03153=1040.366,404.277,-135.134,174.123,44.683,158.891
C03154=1040.356,404.031,-135.089,174.114,44.677,158.888
C03155=1040.347,403.785,-135.044,174.104,44.671,158.886
C03156=1040.337,403.539,-135.000,174.095,44.665,158.884
C03157=1040.327,403.293,-134.955,174.086,44.659,158.881
C03158=1040.318,403.048,-134.910,174.077,44.654,158.879
C03159=1040.309,402.802,-134.864,174.067,44.648,158.876
C03160=1040.299,402.556,-134.820,174.058,44.643,158.874
C03161=1040.290,402.311,-134.776,174.049,44.637,158.872
C03162=1040.280,402.065,-134.731,174.040,44.631,158.869
C03163=1040.270,401.819,-134.687,174.031,44.626,158.867
C03164=1040.261,401.573,-134.642,174.022,44.620,158.865
C03165=1040.251,401.327,-134.598,174.013,44.615,158.862
C03166=1040.242,401.082,-134.553,174.003,44.609,158.860
C03167=1040.232,400.836,-134.509,173.994,44.604,158.858
C03168=1040.223,400.589,-134.465,173.985,44.598,158.855
C03169=1040.214,400.345,-134.420,173.976,44.593,158.853
C03170=1040.204,400.098,-134.376,173.967,44.587,158.851
C03171=1040.195,399.852,-134.332,173.958,44.582,158.849
C03172=1040.185,399.607,-134.287,173.949,44.576,158.846
C03173=1040.176,399.361,-134.243,173.940,44.571,158.844
C03174=1040.166,399.115,-134.199,173.932,44.566,158.842
C03175=1040.158,398.869,-134.155,173.923,44.560,158.840
C03176=1040.148,398.623,-134.111,173.914,44.555,158.837
C03177=1040.139,398.377,-134.067,173.905,44.550,158.835
C03178=1040.130,398.131,-134.023,173.896,44.544,158.833
C03179=1040.120,397.886,-133.980,173.887,44.539,158.831
C03180=1040.110,397.639,-133.936,173.879,44.533,158.829
C03181=1040.102,397.394,-133.892,173.870,44.528,158.826
C03182=1040.092,397.148,-133.848,173.862,44.523,158.824
C03183=1040.083,396.902,-133.804,173.853,44.518,158.822
C03184=1040.074,396.656,-133.760,173.845,44.512,158.820
C03185=1040.065,396.410,-133.716,173.836,44.507,158.818
C03186=1040.055,396.164,-133.673,173.827,44.502,158.816
C03187=1040.046,395.918,-133.629,173.819,44.497,158.813
C03188=1040.037,395.673,-133.586,173.810,44.492,158.811
C03189=1040.028,395.426,-133.542,173.801,44.487,158.809
C03190=1040.019,395.181,-133.498,173.794,44.481,158.807
C03191=1040.009,394.935,-133.455,173.785,44.476,158.805
C03192=1040.001,394.689,-133.412,173.776,44.471,158.803
C03193=1039.991,394.442,-133.368,173.768,44.466,158.801
C03194=1039.983,394.197,-133.325,173.759,44.461,158.799
C03195=1039.973,393.950,-133.282,173.751,44.456,158.797
C03196=1039.964,393.705,-133.238,173.743,44.451,158.794
C03197=1039.955,393.459,-133.195,173.734,44.446,158.792
C03198=1039.946,393.212,-133.152,173.726,44.441,158.790
C03199=1039.937,392.967,-133.109,173.718,44.436,158.788
C03200=1039.928,392.721,-133.066,173.709,44.431,158.786
C03201=1039.920,392.511,-133.029,173.703,44.427,158.784
C03202=1039.912,392.300,-132.992,173.695,44.422,158.783
C03203=1039.904,392.090,-132.956,173.688,44.418,158.781
C03204=1039.897,391.880,-132.919,173.682,44.414,158.779
C03205=1039.889,391.670,-132.882,173.674,44.410,158.778
C03206=1039.882,391.460,-132.845,173.667,44.406,158.776
C03207=1039.874,391.249,-132.809,173.660,44.402,158.774
C03208=1039.866,391.039,-132.772,173.654,44.397,158.772
C03209=1039.857,390.793,-132.729,173.645,44.392,158.770
C03210=1039.849,390.547,-132.686,173.637,44.388,158.768
C03211=1039.839,390.301,-132.644,173.629,44.383,158.767
C03212=1039.831,390.055,-132.601,173.621,44.378,158.764
C03213=1039.821,389.809,-132.558,173.614,44.373,158.763
C03214=1039.813,389.562,-132.516,173.605,44.369,158.761
C03215=1039.803,389.316,-132.473,173.597,44.363,158.759
C03216=1039.795,389.070,-132.430,173.589,44.359,158.757
C03217=1039.786,388.825,-132.388,173.581,44.354,158.755
C03218=1039.778,388.578,-132.345,173.574,44.349,158.753
C03219=1039.768,388.332,-132.303,173.565,44.345,158.751
C03220=1039.760,388.086,-132.260,173.558,44.340,158.749
C03221=1039.751,387.840,-132.218,173.549,44.336,158.747
C03222=1039.742,387.594,-132.176,173.542,44.331,158.745
C03223=1039.733,387.347,-132.133,173.534,44.326,158.743
C03224=1039.724,387.101,-132.091,173.526,44.322,158.741
C03225=1039.715,386.855,-132.049,173.518,44.317,158.739
C03226=1039.706,386.608,-132.007,173.511,44.312,158.738
C03227=1039.696,386.363,-131.965,173.502,44.308,158.736
C03228=1039.688,386.116,-131.923,173.495,44.303,158.734
C03229=1039.679,385.869,-131.881,173.487,44.299,158.732
C03230=1039.670,385.623,-131.839,173.480,44.294,158.730
C03231=1039.662,385.378,-131.797,173.471,44.289,158.728
C03232=1039.654,385.131,-131.755,173.464,44.285,158.726
C03233=1039.645,384.885,-131.713,173.457,44.281,158.725
C03234=1039.636,384.639,-131.671,173.449,44.276,158.723
C03235=1039.627,384.392,-131.630,173.441,44.272,158.721
C03236=1039.618,384.146,-131.588,173.433,44.267,158.719
C03237=1039.610,383.899,-131.546,173.426,44.263,158.717
C03238=1039.601,383.654,-131.504,173.419,44.258,158.715
C03239=1039.592,383.407,-131.462,173.411,44.254,158.714
C03240=1039.583,383.161,-131.421,173.403,44.250,158.712
C03241=1039.575,382.915,-131.379,173.396,44.245,158.710
C03242=1039.566,382.668,-131.337,173.388,44.241,158.708
C03243=1039.558,382.422,-131.295,173.381,44.236,158.707
C03244=1039.549,382.176,-131.254,173.374,44.232,158.705
C03245=1039.540,381.929,-131.212,173.366,44.228,158.703
C03246=1039.532,381.684,-131.171,173.359,44.223,158.701
C03247=1039.524,381.436,-131.129,173.352,44.219,158.700
C03248=1039.515,381.190,-131.087,173.344,44.215,158.698
C03249=1039.507,380.944,-131.046,173.336,44.211,158.696
C03250=1039.498,380.697,-131.005,173.329,44.207,158.694
C03251=1039.489,380.451,-130.963,173.321,44.202,158.692
C03252=1039.481,380.205,-130.922,173.314,44.198,158.691
C03253=1039.473,379.958,-130.880,173.307,44.193,158.689
C03254=1039.465,379.712,-130.839,173.300,44.189,158.687
C03255=1039.456,379.465,-130.798,173.292,44.185,158.686
C03256=1039.448,379.220,-130.757,173.285,44.181,158.684
C03257=1039.439,378.973,-130.716,173.278,44.177,158.682
C03258=1039.431,378.727,-130.674,173.271,44.172,158.681
C03259=1039.422,378.480,-130.633,173.264,44.168,158.679
C03260=1039.414,378.235,-130.592,173.256,44.164,158.677
C03261=1039.401,377.847,-130.528,173.245,44.158,158.675
C03262=1039.387,377.462,-130.463,173.235,44.151,158.672
C03263=1039.374,377.075,-130.400,173.223,44.145,158.669
C03264=1039.360,376.689,-130.336,173.212,44.139,158.667
C03265=1039.352,376.443,-130.295,173.205,44.135,158.665
C03266=1039.344,376.196,-130.254,173.198,44.131,158.664
C03267=1039.335,375.950,-130.214,173.191,44.127,158.662
C03268=1039.327,375.704,-130.173,173.183,44.122,158.660
C03269=1039.318,375.457,-130.132,173.177,44.119,158.659
C03270=1039.310,375.210,-130.092,173.170,44.114,158.657
C03271=1039.302,374.964,-130.051,173.163,44.111,158.656
C03272=1039.294,374.717,-130.010,173.156,44.106,158.654
C03273=1039.285,374.471,-129.970,173.149,44.103,158.652
C03274=1039.277,374.225,-129.929,173.142,44.099,158.651
C03275=1039.268,373.978,-129.888,173.135,44.095,158.649
C03276=1039.260,373.731,-129.848,173.129,44.091,158.648
C03277=1039.252,373.485,-129.808,173.122,44.087,158.646
C03278=1039.244,373.239,-129.768,173.115,44.083,158.644
C03279=1039.235,372.992,-129.727,173.108,44.079,158.643
C03280=1039.227,372.745,-129.687,173.101,44.076,158.641
C03281=1039.219,372.498,-129.646,173.095,44.071,158.640
C03282=1039.211,372.252,-129.606,173.088,44.068,158.638
C03283=1039.203,372.006,-129.566,173.081,44.064,158.637
C03284=1039.194,371.759,-129.525,173.074,44.060,158.635
C03285=1039.186,371.512,-129.485,173.068,44.056,158.634
C03286=1039.178,371.265,-129.445,173.061,44.053,158.632
C03287=1039.170,371.019,-129.404,173.054,44.048,158.630
C03288=1039.162,370.772,-129.365,173.047,44.045,158.629
C03289=1039.154,370.526,-129.324,173.041,44.041,158.627
C03290=1039.146,370.279,-129.284,173.034,44.037,158.626
C03291=1039.138,370.032,-129.244,173.027,44.034,158.624
C03292=1039.129,369.786,-129.204,173.021,44.030,158.623
C03293=1039.121,369.539,-129.164,173.014,44.027,158.622
C03294=1039.113,369.292,-129.125,173.007,44.023,158.620
C03295=1039.104,369.046,-129.085,173.000,44.019,158.619
C03296=1039.096,368.799,-129.045,172.994,44.015,158.617
C03297=1039.088,368.553,-129.005,172.987,44.012,158.616
C03298=1039.080,368.306,-128.965,172.980,44.008,158.614
C03299=1039.072,368.059,-128.926,172.975,44.005,158.613
C03300=1039.064,367.812,-128.886,172.968,44.001,158.611
C03301=1039.056,367.566,-128.847,172.961,43.997,158.610
C03302=1039.048,367.319,-128.807,172.955,43.994,158.608
C03303=1039.039,367.072,-128.768,172.948,43.990,158.607
C03304=1039.032,366.825,-128.728,172.941,43.987,158.605
C03305=1039.023,366.579,-128.688,172.935,43.983,158.604
C03306=1039.016,366.332,-128.648,172.929,43.980,158.602
C03307=1039.007,366.085,-128.609,172.923,43.976,158.601
C03308=1038.999,365.839,-128.570,172.916,43.973,158.600
C03309=1038.991,365.592,-128.530,172.910,43.969,158.598
C03310=1038.983,365.346,-128.491,172.903,43.965,158.597
C03311=1038.975,365.099,-128.451,172.896,43.962,158.595
C03312=1038.967,364.852,-128.412,172.891,43.958,158.594
C03313=1038.959,364.605,-128.372,172.884,43.955,158.593
C03314=1038.951,364.358,-128.333,172.878,43.951,158.591
C03315=1038.944,364.112,-128.294,172.871,43.948,158.590
C03316=1038.936,363.865,-128.255,172.865,43.944,158.588
C03317=1038.924,363.499,-128.196,172.856,43.939,158.586
C03318=1038.912,363.132,-128.139,172.846,43.935,158.584
C03319=1038.901,362.767,-128.080,172.838,43.930,158.582
C03320=1038.889,362.400,-128.022,172.828,43.924,158.580
C03321=1038.881,362.154,-127.983,172.822,43.921,158.579
C03322=1038.873,361.907,-127.944,172.815,43.917,158.577
C03323=1038.865,361.660,-127.905,172.810,43.914,158.576
C03324=1038.857,361.413,-127.866,172.803,43.911,158.575
C03325=1038.850,361.167,-127.827,172.797,43.908,158.573
C03326=1038.841,360.920,-127.788,172.791,43.904,158.572
C03327=1038.833,360.672,-127.749,172.785,43.901,158.571
C03328=1038.825,360.426,-127.710,172.778,43.898,158.569
C03329=1038.817,360.179,-127.672,172.773,43.895,158.568
C03330=1038.809,359.932,-127.633,172.767,43.891,158.567
C03331=1038.802,359.685,-127.594,172.760,43.888,158.566
C03332=1038.794,359.438,-127.556,172.754,43.885,158.564
C03333=1038.786,359.192,-127.517,172.748,43.882,158.563
C03334=1038.778,358.945,-127.478,172.742,43.878,158.562
C03335=1038.770,358.698,-127.440,172.736,43.875,158.560
C03336=1038.762,358.451,-127.401,172.730,43.872,158.559
C03337=1038.754,358.204,-127.363,172.724,43.869,158.558
C03338=1038.747,357.957,-127.324,172.718,43.866,158.556
C03339=1038.739,357.710,-127.286,172.712,43.862,158.555
C03340=1038.731,357.464,-127.248,172.706,43.859,158.554
C03341=1038.724,357.216,-127.208,172.700,43.856,158.553
C03342=1038.716,356.970,-127.170,172.694,43.853,158.551
C03343=1038.708,356.722,-127.132,172.688,43.850,158.550
C03344=1038.700,356.476,-127.093,172.682,43.847,158.549
C03345=1038.692,356.229,-127.055,172.676,43.843,158.547
C03346=1038.685,355.982,-127.016,172.671,43.841,158.546
C03347=1038.677,355.734,-126.979,172.664,43.837,158.545
C03348=1038.669,355.488,-126.940,172.659,43.835,158.544
C03349=1038.661,355.241,-126.902,172.653,43.831,158.543
C03350=1038.653,354.994,-126.864,172.646,43.828,158.541
C03351=1038.645,354.747,-126.826,172.641,43.825,158.540
C03352=1038.637,354.500,-126.788,172.635,43.822,158.539
C03353=1038.630,354.254,-126.750,172.630,43.819,158.538
C03354=1038.622,354.006,-126.712,172.623,43.816,158.536
C03355=1038.614,353.759,-126.674,172.618,43.813,158.535
C03356=1038.607,353.513,-126.635,172.612,43.810,158.534
C03357=1038.599,353.265,-126.597,172.606,43.807,158.533
C03358=1038.592,353.018,-126.559,172.600,43.804,158.532
C03359=1038.584,352.772,-126.522,172.594,43.801,158.530
C03360=1038.575,352.524,-126.484,172.589,43.798,158.529
C03361=1038.568,352.277,-126.446,172.583,43.796,158.528
C03362=1038.561,352.031,-126.408,172.577,43.792,158.527
C03363=1038.553,351.783,-126.370,172.571,43.790,158.526
C03364=1038.545,351.536,-126.332,172.566,43.787,158.524
C03365=1038.538,351.289,-126.294,172.560,43.783,158.523
C03366=1038.531,351.042,-126.257,172.555,43.781,158.522
C03367=1038.522,350.795,-126.219,172.548,43.778,158.521
C03368=1038.515,350.548,-126.181,172.543,43.775,158.520
C03369=1038.507,350.301,-126.144,172.537,43.772,158.518
C03370=1038.500,350.054,-126.105,172.532,43.769,158.517
C03371=1038.493,349.807,-126.068,172.526,43.766,158.516
C03372=1038.485,349.559,-126.030,172.521,43.763,158.515
C03373=1038.473,349.201,-125.976,172.513,43.759,158.513
C03374=1038.462,348.840,-125.922,172.505,43.755,158.512
C03375=1038.451,348.480,-125.867,172.496,43.751,158.510
C03376=1038.440,348.120,-125.812,172.487,43.747,158.508
C03377=1038.433,347.873,-125.775,172.482,43.744,158.507
C03378=1038.424,347.625,-125.738,172.477,43.741,158.506
C03379=1038.417,347.378,-125.700,172.471,43.739,158.505
C03380=1038.410,347.131,-125.663,172.466,43.736,158.504
C03381=1038.402,346.884,-125.626,172.461,43.734,158.503
C03382=1038.395,346.637,-125.588,172.455,43.731,158.502
C03383=1038.387,346.390,-125.551,172.450,43.728,158.501
C03384=1038.379,346.143,-125.514,172.444,43.725,158.499
C03385=1038.372,345.896,-125.476,172.439,43.722,158.498
C03386=1038.364,345.649,-125.439,172.432,43.720,158.497
C03387=1038.357,345.402,-125.402,172.427,43.717,158.496
C03388=1038.349,345.154,-125.365,172.422,43.714,158.495
C03389=1038.342,344.907,-125.328,172.416,43.712,158.494
C03390=1038.334,344.660,-125.291,172.411,43.709,158.493
C03391=1038.327,344.413,-125.253,172.406,43.706,158.492
C03392=1038.320,344.166,-125.217,172.400,43.703,158.491
C03393=1038.312,343.919,-125.180,172.395,43.701,158.490
C03394=1038.305,343.672,-125.142,172.390,43.698,158.488
C03395=1038.297,343.424,-125.106,172.384,43.696,158.487
C03396=1038.290,343.177,-125.068,172.379,43.693,158.486
C03397=1038.282,342.930,-125.031,172.374,43.691,158.485
C03398=1038.275,342.682,-124.995,172.368,43.688,158.484
C03399=1038.267,342.436,-124.958,172.363,43.686,158.483
C03400=1038.260,342.189,-124.921,172.358,43.683,158.482
C03401=1038.253,341.942,-124.884,172.352,43.680,158.481
C03402=1038.245,341.694,-124.848,172.347,43.678,158.480
C03403=1038.238,341.447,-124.811,172.342,43.675,158.479
C03404=1038.230,341.200,-124.774,172.336,43.673,158.478
C03405=1038.223,340.952,-124.738,172.331,43.670,158.477
C03406=1038.215,340.705,-124.701,172.326,43.668,158.476
C03407=1038.207,340.458,-124.664,172.320,43.665,158.475
C03408=1038.200,340.211,-124.629,172.315,43.663,158.474
C03409=1038.193,339.964,-124.591,172.310,43.660,158.473
C03410=1038.185,339.716,-124.555,172.306,43.657,158.472
C03411=1038.178,339.469,-124.519,172.300,43.655,158.471
C03412=1038.170,339.222,-124.482,172.295,43.652,158.470
C03413=1038.163,338.975,-124.445,172.290,43.650,158.469
C03414=1038.156,338.728,-124.409,172.284,43.647,158.468
C03415=1038.148,338.480,-124.373,172.279,43.645,158.467
C03416=1038.140,338.233,-124.337,172.274,43.643,158.466
C03417=1038.134,337.986,-124.300,172.269,43.640,158.465
C03418=1038.126,337.739,-124.263,172.263,43.638,158.464
C03419=1038.118,337.491,-124.227,172.258,43.635,158.463
C03420=1038.111,337.244,-124.191,172.253,43.633,158.462
C03421=1038.104,336.997,-124.154,172.249,43.630,158.461
C03422=1038.097,336.749,-124.118,172.244,43.628,158.460
C03423=1038.089,336.502,-124.082,172.238,43.626,158.459
C03424=1038.082,336.255,-124.046,172.233,43.623,158.458
C03425=1038.074,336.008,-124.010,172.228,43.621,158.457
C03426=1038.067,335.760,-123.973,172.223,43.618,158.456
C03427=1038.060,335.513,-123.937,172.217,43.616,158.455
C03428=1038.053,335.266,-123.901,172.213,43.614,158.454
C03429=1038.043,334.902,-123.848,172.205,43.610,158.452
C03430=1038.031,334.539,-123.795,172.198,43.607,158.451
C03431=1038.020,334.175,-123.742,172.191,43.604,158.450
C03432=1038.010,333.812,-123.690,172.183,43.600,158.448
C03433=1038.002,333.564,-123.654,172.178,43.598,158.447
C03434=1037.995,333.316,-123.618,172.173,43.596,158.446
C03435=1037.987,333.070,-123.582,172.169,43.593,158.445
C03436=1037.980,332.822,-123.546,172.164,43.591,158.444
C03437=1037.973,332.575,-123.511,172.158,43.589,158.443
C03438=1037.965,332.327,-123.475,172.153,43.586,158.442
C03439=1037.959,332.080,-123.439,172.148,43.584,158.441
C03440=1037.951,331.833,-123.403,172.144,43.582,158.441
C03441=1037.944,331.586,-123.367,172.139,43.580,158.440
C03442=1037.936,331.338,-123.332,172.134,43.578,158.439
C03443=1037.929,331.091,-123.296,172.129,43.576,158.438
C03444=1037.922,330.843,-123.261,172.123,43.573,158.437
C03445=1037.915,330.596,-123.225,172.119,43.571,158.436
C03446=1037.908,330.348,-123.189,172.114,43.569,158.435
C03447=1037.901,330.101,-123.153,172.109,43.566,158.434
C03448=1037.893,329.853,-123.118,172.105,43.565,158.433
C03449=1037.886,329.607,-123.082,172.100,43.562,158.432
C03450=1037.879,329.359,-123.047,172.095,43.560,158.431
C03451=1037.871,329.112,-123.011,172.089,43.558,158.430
C03452=1037.864,328.865,-122.976,172.085,43.555,158.430
C03453=1037.857,328.617,-122.941,172.080,43.554,158.429
C03454=1037.850,328.369,-122.905,172.075,43.551,158.428
C03455=1037.842,328.123,-122.870,172.070,43.549,158.427
C03456=1037.835,327.875,-122.835,172.066,43.547,158.426
C03457=1037.828,327.627,-122.800,172.061,43.545,158.425
C03458=1037.820,327.380,-122.765,172.056,43.543,158.424
C03459=1037.813,327.132,-122.730,172.051,43.541,158.423
C03460=1037.805,326.885,-122.695,172.047,43.539,158.423
C03461=1037.798,326.638,-122.659,172.042,43.537,158.422
C03462=1037.790,326.391,-122.624,172.037,43.535,158.421
C03463=1037.783,326.143,-122.589,172.033,43.533,158.420
C03464=1037.776,325.896,-122.554,172.028,43.531,158.419
C03465=1037.769,325.648,-122.519,172.023,43.529,158.418
C03466=1037.761,325.401,-122.484,172.019,43.527,158.417
C03467=1037.754,325.153,-122.449,172.013,43.525,158.417
C03468=1037.746,324.906,-122.414,172.008,43.523,158.416
C03469=1037.739,324.658,-122.379,172.004,43.521,158.415
C03470=1037.732,324.411,-122.344,171.999,43.519,158.414
C03471=1037.725,324.164,-122.309,171.994,43.517,158.413
C03472=1037.718,323.916,-122.274,171.990,43.515,158.412
C03473=1037.710,323.668,-122.240,171.985,43.513,158.412
C03474=1037.703,323.421,-122.205,171.980,43.511,158.411
C03475=1037.696,323.173,-122.170,171.976,43.509,158.410
C03476=1037.689,322.926,-122.135,171.971,43.508,158.409
C03477=1037.681,322.678,-122.100,171.966,43.505,158.408
C03478=1037.674,322.431,-122.065,171.962,43.503,158.407
C03479=1037.667,322.183,-122.031,171.957,43.502,158.407
C03480=1037.660,321.936,-121.996,171.953,43.499,158.406
C03481=1037.653,321.689,-121.962,171.948,43.498,158.405
C03482=1037.646,321.442,-121.926,171.943,43.496,158.404
C03483=1037.638,321.193,-121.892,171.939,43.493,158.403
C03484=1037.631,320.946,-121.857,171.934,43.492,158.402
C03485=1037.621,320.578,-121.806,171.928,43.489,158.401
C03486=1037.611,320.210,-121.755,171.921,43.486,158.400
C03487=1037.600,319.841,-121.703,171.914,43.483,158.399
C03488=1037.589,319.473,-121.652,171.907,43.481,158.398
C03489=1037.582,319.226,-121.617,171.902,43.479,158.397
C03490=1037.575,318.979,-121.582,171.898,43.476,158.396
C03491=1037.568,318.731,-121.548,171.893,43.475,158.395
C03492=1037.561,318.484,-121.513,171.889,43.473,158.394
C03493=1037.554,318.236,-121.479,171.885,43.471,158.394
C03494=1037.547,317.989,-121.444,171.881,43.469,158.393
C03495=1037.540,317.741,-121.410,171.876,43.468,158.392
C03496=1037.533,317.494,-121.375,171.872,43.465,158.391
C03497=1037.526,317.246,-121.341,171.867,43.464,158.390
C03498=1037.519,316.998,-121.306,171.863,43.462,158.390
C03499=1037.512,316.751,-121.272,171.858,43.460,158.389
C03500=1037.505,316.503,-121.238,171.854,43.458,158.388
C03501=1037.498,316.256,-121.203,171.849,43.456,158.387
C03502=1037.491,316.008,-121.169,171.845,43.455,158.387
C03503=1037.484,315.761,-121.134,171.840,43.453,158.386
C03504=1037.477,315.513,-121.100,171.836,43.451,158.385
C03505=1037.470,315.265,-121.066,171.831,43.449,158.384
C03506=1037.463,315.019,-121.032,171.827,43.447,158.383
C03507=1037.457,314.771,-120.997,171.822,43.445,158.383
C03508=1037.450,314.523,-120.964,171.818,43.443,158.382
C03509=1037.442,314.276,-120.929,171.813,43.442,158.381
C03510=1037.436,314.028,-120.895,171.809,43.440,158.380
C03511=1037.428,313.780,-120.861,171.805,43.438,158.380
C03512=1037.422,313.532,-120.826,171.800,43.436,158.379
C03513=1037.415,313.286,-120.792,171.797,43.434,158.378
C03514=1037.409,313.038,-120.758,171.792,43.433,158.377
C03515=1037.401,312.790,-120.724,171.788,43.431,158.377
C03516=1037.394,312.543,-120.690,171.783,43.429,158.376
C03517=1037.388,312.295,-120.656,171.779,43.427,158.375
C03518=1037.381,312.048,-120.622,171.775,43.425,158.374
C03519=1037.374,311.800,-120.587,171.770,43.424,158.374
C03520=1037.367,311.552,-120.555,171.766,43.422,158.373
C03521=1037.360,311.305,-120.521,171.761,43.421,158.372
C03522=1037.352,311.057,-120.487,171.757,43.419,158.371
C03523=1037.346,310.810,-120.454,171.753,43.418,158.371
C03524=1037.339,310.562,-120.420,171.749,43.416,158.370
C03525=1037.331,310.315,-120.386,171.745,43.414,158.369
C03526=1037.323,310.067,-120.353,171.740,43.413,158.369
C03527=1037.316,309.820,-120.319,171.736,43.411,158.368
C03528=1037.309,309.571,-120.286,171.731,43.409,158.367
C03529=1037.303,309.324,-120.252,171.728,43.408,158.366
C03530=1037.296,309.077,-120.218,171.723,43.406,158.366
C03531=1037.288,308.829,-120.185,171.719,43.405,158.365
C03532=1037.281,308.581,-120.152,171.715,43.403,158.364
C03533=1037.274,308.334,-120.119,171.710,43.401,158.364
C03534=1037.267,308.086,-120.085,171.707,43.400,158.363
C03535=1037.260,307.839,-120.051,171.702,43.398,158.362
C03536=1037.253,307.590,-120.018,171.698,43.397,158.362
C03537=1037.246,307.344,-119.984,171.694,43.395,158.361
C03538=1037.238,307.096,-119.951,171.689,43.394,158.360
C03539=1037.231,306.848,-119.918,171.685,43.392,158.360
C03540=1037.225,306.601,-119.885,171.680,43.391,158.359
C03541=1037.214,306.237,-119.836,171.675,43.388,158.358
C03542=1037.204,305.874,-119.787,171.669,43.386,158.357
C03543=1037.194,305.510,-119.738,171.663,43.384,158.356
C03544=1037.184,305.147,-119.689,171.657,43.382,158.355
C03545=1037.177,304.899,-119.655,171.652,43.380,158.354
C03546=1037.169,304.651,-119.623,171.648,43.379,158.353
C03547=1037.162,304.404,-119.590,171.644,43.377,158.353
C03548=1037.155,304.156,-119.556,171.640,43.376,158.352
C03549=1037.149,303.908,-119.524,171.636,43.374,158.351
C03550=1037.142,303.661,-119.490,171.632,43.373,158.351
C03551=1037.135,303.413,-119.458,171.628,43.371,158.350
C03552=1037.128,303.166,-119.424,171.623,43.370,158.349
C03553=1037.121,302.917,-119.391,171.620,43.369,158.349
C03554=1037.114,302.671,-119.357,171.616,43.367,158.348
C03555=1037.107,302.423,-119.325,171.611,43.366,158.347
C03556=1037.100,302.175,-119.292,171.607,43.364,158.347
C03557=1037.093,301.927,-119.258,171.603,43.362,158.346
C03558=1037.087,301.680,-119.225,171.600,43.360,158.345
C03559=1037.080,301.431,-119.192,171.595,43.359,158.345
C03560=1037.073,301.185,-119.160,171.591,43.358,158.344
C03561=1037.066,300.936,-119.126,171.587,43.356,158.343
C03562=1037.059,300.689,-119.094,171.583,43.355,158.343
C03563=1037.053,300.441,-119.061,171.579,43.354,158.342
C03564=1037.045,300.194,-119.028,171.575,43.352,158.342
C03565=1037.039,299.946,-118.995,171.571,43.351,158.341
C03566=1037.032,299.698,-118.962,171.568,43.349,158.340
C03567=1037.026,299.450,-118.929,171.563,43.348,158.340
C03568=1037.018,299.202,-118.897,171.559,43.346,158.339
C03569=1037.011,298.955,-118.863,171.555,43.345,158.338
C03570=1037.005,298.708,-118.830,171.551,43.343,158.338
C03571=1036.998,298.460,-118.797,171.547,43.342,158.337
C03572=1036.991,298.212,-118.765,171.543,43.341,158.336
C03573=1036.984,297.964,-118.732,171.539,43.339,158.336
C03574=1036.978,297.716,-118.699,171.535,43.338,158.335
C03575=1036.972,297.469,-118.667,171.532,43.336,158.335
C03576=1036.964,297.221,-118.634,171.527,43.335,158.334
C03577=1036.958,296.973,-118.601,171.523,43.333,158.333
C03578=1036.952,296.726,-118.569,171.519,43.332,158.333
C03579=1036.945,296.477,-118.535,171.516,43.331,158.332
C03580=1036.938,296.230,-118.503,171.512,43.329,158.331
C03581=1036.931,295.982,-118.471,171.508,43.327,158.331
C03582=1036.924,295.734,-118.437,171.503,43.326,158.330
C03583=1036.918,295.487,-118.405,171.500,43.325,158.329
C03584=1036.911,295.239,-118.373,171.496,43.323,158.329
C03585=1036.905,294.992,-118.340,171.492,43.322,158.328
C03586=1036.897,294.744,-118.307,171.488,43.321,158.328
C03587=1036.891,294.496,-118.275,171.485,43.319,158.327
C03588=1036.884,294.249,-118.242,171.480,43.318,158.326
C03589=1036.877,294.000,-118.210,171.476,43.317,158.326
C03590=1036.870,293.753,-118.178,171.473,43.316,158.325
C03591=1036.863,293.505,-118.146,171.469,43.314,158.325
C03592=1036.856,293.257,-118.113,171.465,43.313,158.324
C03593=1036.850,293.009,-118.081,171.462,43.312,158.323
C03594=1036.843,292.762,-118.048,171.457,43.311,158.323
C03595=1036.836,292.514,-118.016,171.453,43.309,158.322
